(* CODESYS project Tc3_UnitTest.library
   Description: Twincat 3 unit test library
   Version: 1.0.0.4
   Title: Tc3_UnitTest
   Company: Zerlauth
   DocFormat: TcDocGen
   Placeholder: Tc3_UnitTest
   Author: www.peterzerlauth.com
   DefaultNamespace: Tc3_UnitTest

Project tree, tasks and I/O mapping:
  libraries: Tc2_Standard, * (Beckhoff Automation GmbH); Tc2_System, * (Beckhoff Automation GmbH); Tc2_Utilities, * (Beckhoff Automation GmbH); Tc3_JsonXml, * (Beckhoff Automation GmbH); Tc3_Module, * (Beckhoff Automation GmbH)
  Assert/
    data type E_AdsError
    data type E_Assert
    function block FB_Assert [ST]: M_Assert, M_Equals, M_Equals_Array_LREAL, M_Equals_Array_REAL, M_Equals_BOOL, M_Equals_BYTE, M_Equals_DINT, M_Equals_INT, M_Equals_LINT, M_Equals_LREAL, M_Equals_REAL, M_Equals_STRING, M_Equals_TIME, M_Equals_UDINT, M_Equals_UINT, M_Equals_ULINT, M_Equals_UXINT, M_Equals_WSTRING, M_Equals_XINT, M_Equals_XWORD, M_Error, M_Failure, M_IsTRUE, M_Passed, M_Reset, M_Skip
    interface I_Assert: M_Assert, M_Equals, M_Equals_Array_LREAL, M_Equals_Array_REAL, M_Equals_BOOL, M_Equals_BYTE, M_Equals_DINT, M_Equals_INT, M_Equals_LINT, M_Equals_LREAL, M_Equals_REAL, M_Equals_STRING, M_Equals_TIME, M_Equals_UDINT, M_Equals_UINT, M_Equals_ULINT, M_Equals_UXINT, M_Equals_WSTRING, M_Equals_XINT, M_Equals_XWORD, M_Error, M_Failure, M_IsTRUE, M_Passed, M_Reset, M_Skip
  Base/
    data type E_Base
    function F_GetCycleTime [ST]
    function F_GetName [ST]
    function block FB_Base [ST]: M_Aborted, M_Aborting, M_Execute, M_Init, M_Request, M_Starting, M_Stopped, M_Stopping, P_State
    interface I_Base: M_Request, P_State
  File/
    function block FB_File [ST]: M_Append, M_AppendLine, M_Close, M_Create, M_Delete, M_Load, M_Open, M_Read, M_Write, P_Error
    interface I_File: M_Append, M_AppendLine, M_Close, M_Create, M_Delete, M_Load, M_Open, M_Read, M_Write, P_Error
  List/
    Builder/
      function block FB_StringBuilder [ST]: FB_exit, M_Append, M_AppendBOOL, M_AppendINT, M_AppendREAL, M_Contains, M_Find, M_Insert, M_Reset, M_ToAny, M_ToString, P_Length
      interface I_StringBuilder: M_Append, M_AppendBOOL, M_AppendINT, M_AppendREAL, M_Contains, M_Find, M_Insert, M_Reset, M_ToAny, M_ToString, P_Length
    Object/
      function block FB_ListObject [ST]: FB_exit, M_Add, M_Clear, M_Find, M_Get, M_Index, M_Remove, P_Length
      interface I_ListObject: M_Add, M_Clear, M_Find, M_Get, M_Index, M_Remove, P_Length
      interface I_Object
    String/
      function block FB_ListSTRING [ST]: FB_exit, M_Add, M_Clear, M_Find, M_Index, M_Insert, M_Item, M_Remove, M_Set, P_Length
      interface I_ListSTRING: M_Add, M_Clear, M_Find, M_Index, M_Insert, M_Item, M_Remove, M_Set, P_Length
  Logger/
    data type E_LogLevel
    function block FB_Logger [ST]: M_Critical, M_Debug, M_Error, M_Info, M_Log, M_Warning, P_Settings
    function block FB_TcLogger [ST]: M_Critical, M_Debug, M_Error, M_Info, M_Log, M_Warning, P_Settings
    interface I_Logger: M_Critical, M_Debug, M_Error, M_Info, M_Log, M_Warning, P_Settings
    data type ST_LoggerSettings
  Property/
    function block FB_Property [ST]: M_Add, M_Reset, P_List
    interface I_Property: M_Add, M_Reset
  Testcase/
    data type E_Testcase
    data type ST_Testcase
  Testsuite/
    function block FB_Testsuite [ST]: M_Execute, M_Starting, M_Stopping, M_Testcase, P_Assert, P_File, P_List, P_Logger, P_Options, P_Parent, P_Property, P_Testcase
    interface I_Testsuite: P_File, P_List, P_Logger, P_Options, P_Parent, P_Testcase
    data type ST_Testsuite
    data type ST_TestsuiteOptions
  Testsuites/
    function block FB_Testsuites [ST]: M_Add, M_Execute, M_Starting, M_Stopping, P_Data, P_List, P_Options, P_Property
    interface I_Testsuites: P_Data, P_List, P_Options, P_Property
    data type ST_Testsuites
    data type ST_TestsuitesOptions
  Version/
    global variables Global_Version
*)

// Assert/E_AdsError
{attribute 'qualified_only'}
{attribute 'to_string'}
TYPE E_AdsError :
(
	NOERR:= 0,
	ROUTER_NOLOCKEDMEMORY:= 1280,
	ROUTER_RESIZEMEMORY:= 1281,
	ROUTER_MAILBOXFULL:= 1282,
	ROUTER_DEBUGBOXFULL:= 1283,
	ROUTER_UNKNOWNPORTTYPE:= 1284,
	ROUTER_NOTINITIALIZED:= 1285,
	ROUTER_PORTALREADYINUSE:= 1286,
	ROUTER_NOTREGISTERED:= 1287,
	ROUTER_NOMOREQUEUES:= 1288,
	ROUTER_INVALIDPORT:= 1289,
	ROUTER_NOTACTIVATED:= 1290,
	ROUTER_FRAGMENTBOXFULL:= 1291,
	ROUTER_FRAGMENTTIMEOUT:= 1292,
	ROUTER_TOBEREMOVED:= 1293,
	DEVICE_ERROR:= 1792,
	DEVICE_SRVNOTSUPP:= 1793,
	DEVICE_INVALIDGRP:= 1794,
	DEVICE_INVALIDOFFSET:= 1795,
	DEVICE_INVALIDACCESS:= 1796,
	DEVICE_INVALIDSIZE:= 1797,
	DEVICE_INVALIDDATA:= 1798,
	DEVICE_NOTREADY:= 1799,
	DEVICE_BUSY:= 1800,
	DEVICE_INVALIDCONTEXT:= 1801,
	DEVICE_NOMEMORY:= 1802,
	DEVICE_INVALIDPARM:= 1803,
	DEVICE_NOTFOUND:= 1804,
	DEVICE_SYNTAX:= 1805,
	DEVICE_INCOMPATIBLE:= 1806,
	DEVICE_EXISTS:= 1807,
	DEVICE_SYMBOLNOTFOUND:= 1808,
	DEVICE_SYMBOLVERSIONINVALID:= 1809,
	DEVICE_INVALIDSTATE:= 1810,
	DEVICE_TRANSMODENOTSUPP:= 1811,
	DEVICE_NOTIFYHNDINVALID:= 1812,
	DEVICE_CLIENTUNKNOWN:= 1813,
	DEVICE_NOMOREHDLS:= 1814,
	DEVICE_INVALIDWATCHSIZE:= 1815,
	DEVICE_NOTINIT:= 1816,
	DEVICE_TIMEOUT:= 1817,
	DEVICE_NOINTERFACE:= 1818,
	DEVICE_INVALIDINTERFACE:= 1819,
	DEVICE_INVALIDCLSID:= 1820,
	DEVICE_INVALIDOBJID:= 1821,
	DEVICE_PENDING:= 1822,
	DEVICE_ABORTED:= 1823,
	DEVICE_WARNING:= 1824,
	DEVICE_INVALIDARRAYIDX:= 1825,
	DEVICE_SYMBOLNOTACTIVE:= 1826,
	DEVICE_ACCESSDENIED:= 1827,
	DEVICE_LICENSENOTFOUND:= 1828,
	DEVICE_LICENSEEXPIRED:= 1829,
	DEVICE_LICENSEEXCEEDED:= 1830,
	DEVICE_LICENSEINVALID:= 1831,
	DEVICE_LICENSESYSTEMID:= 1832,
	DEVICE_LICENSENOTIMELIMIT:= 1833,
	DEVICE_LICENSEFUTUREISSUE:= 1834,
	DEVICE_LICENSETIMETOLONG:= 1835,
	DEVICE_EXCEPTION:= 1836,
	DEVICE_LICENSEDUPLICATED:= 1837,
	CLIENT_ERROR:= 1856,
	CLIENT_INVALIDPARM:= 1857,
	CLIENT_LISTEMPTY:= 1858,
	CLIENT_VARUSED:= 1859,
	CLIENT_DUPLINVOKEID:= 1860,
	CLIENT_SYNCTIMEOUT:= 1861,
	CLIENT_W32ERROR:= 1862,
	CLIENT_TIMEOUTINVALID:= 1863,
	CLIENT_PORTNOTOPEN:= 1864,
	CLIENT_NOAMSADDR:= 1865,
	CLIENT_SYNCINTERNAL:= 1872,
	CLIENT_ADDHASH:= 1873,
	CLIENT_REMOVEHASH:= 1874,
	CLIENT_NOMORESYM:= 1875,
	CLIENT_SYNCRESINVALID:= 1876,
	CLIENT_SYNCPORTLOCKED:= 1877
)UDINT;
END_TYPE

// Assert/E_Assert
{attribute 'qualified_only'}
{attribute 'strict'}
TYPE E_Assert :
(
	Passed	:= 0,
	Failure	:= 1,
	Error	:= 2,
	Skipped	:= 3
)USINT;
END_TYPE

// Base/E_Base
{attribute 'qualified_only'}
{attribute 'strict'}
TYPE E_Base :
(
	{attribute 'hide'} 
	Init 	:= 0,
	Starting:= 2,	
	Execute	:= 3,
	Stopping:= 4,
	Aborting:= 5,
	Aborted	:= 6,
	Reset	:= 7,
	Stopped	:= 1
)USINT;
END_TYPE

// Logger/E_LogLevel
{attribute 'qualified_only'}
{attribute 'strict'}
TYPE E_LogLevel :
(
	Debug:=		0, 
    Info:= 		1, 
    Warning:= 	2, 
    Error:= 	3, 
    Critical:= 	4
);
END_TYPE

// Logger/ST_LoggerSettings
TYPE ST_LoggerSettings :
STRUCT
	eLogLevelMinimum:		E_LogLevel:= E_LogLevel.Debug;
	eLogLevelMaximum:		E_LogLevel:= E_LogLevel.Critical;
END_STRUCT
END_TYPE

// Testcase/E_Testcase
{attribute 'qualified_only'}
{attribute 'strict'}
TYPE E_Testcase :
(
	Init    := -32768,
	Start 	:= 0,
	Done	:= 32767
)INT;
END_TYPE

// Testcase/ST_Testcase
TYPE ST_Testcase :
STRUCT
	sName:				STRING(255);	//	name        The name of this test case, often the method name  
	sClassname:			STRING(255);	//	classname   The name of the parent class/folder, often the same as the suite's name
	nAssertions:		DINT; 			//	assertions  Number of assertions checked during test case execution  
	fTime:				LREAL;			//	time        Execution time of the test in seconds            
	sFile:				STRING(255);	//	file        Source code file of this test case              
	sLine:				STRING(255);	//	line        Source code line number of the start of this test case  
END_STRUCT
END_TYPE

// Testsuite/ST_Testsuite
TYPE ST_Testsuite :
STRUCT
	sName:				STRING(255):= 'testsuite'; 	// Name OF the entire test run
	nTests:				DINT;						// tests       Total number of tests in this suite          
	nFailures:			DINT;						// failures    Total number of failed tests in this suite   
	nErrors:			DINT;						// errors      Total number of errored tests in this suite 
	nSkipped:			DINT;						// skipped     Total number of skipped tests in this suite            
	nAssertions:		DINT;						// assertions  Total number of assertions for all tests in this suite  
	fTime: 				LREAL;						// time        Aggregated time of all tests in this file in seconds  (100ns)   
	sTimestamp:			STRING(39);					// timestamp   Date and time of when the test suite was executed (in ISO 8601 format)  
	sFile:				STRING(255);				// file        Source code file of this test suite
END_STRUCT
END_TYPE

// Testsuite/ST_TestsuiteOptions
TYPE ST_TestsuiteOptions :
STRUCT
		bAbortOnError:			BOOL;
END_STRUCT
END_TYPE

// Testsuites/ST_Testsuites
TYPE ST_Testsuites :
STRUCT
	sName:				STRING(255); 				// Name OF the entire test run
	nTests:				DINT;						// Total number of tests in this file
	nFailures:			dINT;						// Total number of failed tests in this file
	nErrors:			dINT;						// Total number of errored tests in this file
	nSkipped:			dINT;						// Total number of skipped tests in this file
	nAssertions:		dINT;						// Total number of assertions for all tests in this file
	fTime:				LREAL;						// Aggregated time of all tests in this file in seconds
	sTimestamp:			STRING(39);					// timestamp   Date and time of when the test suite was executed (in ISO 8601 format)
END_STRUCT
END_TYPE

// Testsuites/ST_TestsuitesOptions
TYPE ST_TestsuitesOptions :
STRUCT
	sFilePathName:		STRING(255):= 'C:\report.xml';		// as Property
END_STRUCT
END_TYPE

// Version/Global_Version
{attribute 'TcGenerated'}
{attribute 'no-analysis'}
{attribute 'linkalways'}
// This function has been automatically generated from the project information.
VAR_GLOBAL CONSTANT
	{attribute 'const_non_replaced'}
	stLibVersion_Tc3_UnitTest : ST_LibVersion := (iMajor := 1, iMinor := 0, iBuild := 0, iRevision := 4, nFlags := 0, sVersion := '1.0.0.4');
END_VAR

// Assert/FB_Assert
FUNCTION_BLOCK FB_Assert IMPLEMENTS I_Assert
VAR_INPUT
END_VAR
VAR_OUTPUT
	fbList:					FB_ListSTRING;
	nAssert:				DINT;
	nPassed:				DINT;
	nSkipped:				DINT;
	nFailures:				DINT;
	nErrors:				DINT;
END_VAR
VAR
	fbJson:					FB_JsonSaxWriter;
  	fbJsonDataType:			FB_JsonReadWriteDataType;
	fbBuilder:				FB_StringBuilder;
END_VAR

METHOD PUBLIC M_Assert
VAR_INPUT
END_VAR
IF nSkipped = 0 THEN
	nAssert:= nAssert + 1;
END_IF
END_METHOD

METHOD PUBLIC M_Equals : I_Assert
VAR_INPUT
	Expected:			ANY;			// Expected as udint
    Actual:				ANY;          	// Actual as udint
	Message:			STRING(255);   	// Message as string
END_VAR
VAR
	sJsonExpected:			STRING(2000);
	sJsonActual:			STRING(2000); 
	sDatatypeExpected:		STRING(255); 
	sDatatypeActual:		STRING(255);
END_VAR
M_Assert();

fbJson.ResetDocument();
sDatatypeExpected:= fbJsonDataType.GetDatatypeNameByAddress(nData:= DINT_TO_UDINT(Expected.diSize), pData:= Expected.pValue);
fbJsonDataType.AddJsonValueFromSymbol(fbJson, sDatatypeExpected, DINT_TO_UDINT(Expected.diSize), Expected.pValue);
fbJson.CopyDocument(sJsonExpected, SIZEOF(sJsonExpected));

fbJson.ResetDocument();
sDatatypeActual:= fbJsonDataType.GetDatatypeNameByAddress(nData:= DINT_TO_UDINT(Actual.diSize), pData:= Actual.pValue);
fbJsonDataType.AddJsonValueFromSymbol(fbJson, sDatatypeActual, DINT_TO_UDINT(Actual.diSize), Actual.pValue);
fbJson.CopyDocument(sJsonActual, SIZEOF(sJsonActual));

IF sDatatypeExpected <> sDatatypeActual THEN
	fbBuilder.M_Reset();
	fbBuilder.M_Append('Expected = ');
	fbBuilder.M_Append(sDatatypeExpected);
	fbBuilder.M_Append(' Actual = ');
	fbBuilder.M_Append(sDatatypeActual);
	M_Failure(fbBuilder.M_ToString(), Message);
ELSIF sJsonExpected <> sJsonActual THEN
	fbBuilder.M_Reset();
	fbBuilder.M_Append('Expected = ');
	fbBuilder.M_Append(sJsonExpected);
	fbBuilder.M_Append(' Actual = ');
	fbBuilder.M_Append(sJsonActual);
	M_Failure(fbBuilder.M_ToString(), Message);
END_IF
M_Equals:= THIS^;
END_METHOD

METHOD PUBLIC M_Equals_Array_LREAL : I_Assert
VAR_IN_OUT
	Expected:			ARRAY [*] OF LREAL;	// Expected as array of lreal
	Actual:				ARRAY [*] OF LREAL;	// Actual as array of lreal
END_VAR                                    
VAR_INPUT                                  
	Tolerance:			LREAL;              // Tolerance as lreal
	Message:			STRING(255);		// Message as string
END_VAR

VAR
	nIndex:				DINT;
END_VAR
M_Equals_Array_LREAL:= THIS^;
M_Assert();
IF LOWER_BOUND(Expected, 1) <> LOWER_BOUND(Actual, 1) THEN
	M_Failure('', Message);
ELSIF UPPER_BOUND(Expected, 1) <> UPPER_BOUND(Actual, 1) THEN
	M_Failure('', Message);
ELSE
	FOR nIndex:= LOWER_BOUND(Expected, 1) TO UPPER_BOUND(Expected, 1) DO
		IF ABS(Expected[nIndex] - Actual[nIndex]) > ABS(Tolerance) THEN	
			fbBuilder.M_Reset();
			fbBuilder.M_Append('Index = [');
			fbBuilder.M_Append(DINT_TO_STRING(nIndex));
			fbBuilder.M_Append('] Expected = ]');
			fbBuilder.M_Append(LREAL_TO_STRING(Expected[nIndex]));
			fbBuilder.M_Append('] Actual = [');
			fbBuilder.M_Append(LREAL_TO_STRING(Actual[nIndex]));
			fbBuilder.M_Append('] Tolerance = ]');
			fbBuilder.M_Append(LREAL_TO_STRING(Tolerance));
			fbBuilder.M_Append(']');
			M_Failure(fbBuilder.M_ToString(), Message);
			RETURN;
		END_IF
	END_FOR
	M_Passed();
END_IF
END_METHOD

METHOD PUBLIC M_Equals_Array_REAL : I_Assert
VAR_IN_OUT
	Expected:			ARRAY [*] OF REAL;	// Expected as array of real
	Actual:				ARRAY [*] OF REAL;	// Actual as array of real
END_VAR                                   
VAR_INPUT                                 
	Tolerance:			REAL;             	// Tolerance as real
	Message:			STRING(255);      	// Message as string
END_VAR

VAR
	nIndex:				DINT;
END_VAR
M_Equals_Array_REAL:= THIS^;
M_Assert();
IF LOWER_BOUND(Expected, 1) <> LOWER_BOUND(Actual, 1) THEN
	M_Failure('', Message);
ELSIF UPPER_BOUND(Expected, 1) <> UPPER_BOUND(Actual, 1) THEN
	M_Failure('', Message);
ELSE
	FOR nIndex:= LOWER_BOUND(Expected, 1) TO UPPER_BOUND(Expected, 1) DO
		IF ABS(Expected[nIndex] - Actual[nIndex]) > ABS(Tolerance) THEN	
			fbBuilder.M_Reset();
			fbBuilder.M_Append('Index = [');
			fbBuilder.M_Append(DINT_TO_STRING(nIndex));
			fbBuilder.M_Append('] Expected = ]');
			fbBuilder.M_Append(REAL_TO_STRING(Expected[nIndex]));
			fbBuilder.M_Append('] Actual = "');
			fbBuilder.M_Append(REAL_TO_STRING(Actual[nIndex]));
			fbBuilder.M_Append('] Tolerance = [');
			fbBuilder.M_Append(REAL_TO_STRING(Tolerance));
			fbBuilder.M_Append(']');
			M_Failure(fbBuilder.M_ToString(), Message);
			RETURN;
		END_IF
	END_FOR
	M_Passed();
END_IF
END_METHOD

METHOD PUBLIC M_Equals_BOOL : I_Assert
VAR_INPUT
	Expected:			BOOL;				// Expected as bool
    Actual:				BOOL;           	// Actual as bool
	Message:			STRING(255);    	// Message as string
END_VAR
M_Assert();
IF Expected = Actual THEN
	M_Passed();
ELSE
	fbBuilder.M_Reset();
	fbBuilder.M_Append('Expected = [');
	fbBuilder.M_Append(BOOL_TO_STRING(Expected));
	fbBuilder.M_Append('] Actual = [');
	fbBuilder.M_Append(BOOL_TO_STRING(Actual));
	fbBuilder.M_Append(']');
	M_Failure(fbBuilder.M_ToString(), Message);
END_IF
M_Equals_BOOL:= THIS^;
END_METHOD

METHOD PUBLIC M_Equals_BYTE : I_Assert
VAR_INPUT
	Expected:			BYTE;			// Expected as byte
    Actual:				BYTE;           // Actual as byte
	Message:			STRING(255);    // Message as string
END_VAR
M_Assert();
IF Expected = Actual THEN
	M_Passed();
ELSE
	fbBuilder.M_Reset();
	fbBuilder.M_Append('Expected = [');
	fbBuilder.M_Append(BYTE_TO_STRING(Expected));
	fbBuilder.M_Append('] Actual = [');
	fbBuilder.M_Append(BYTE_TO_STRING(Actual));
	fbBuilder.M_Append(']');
	M_Failure(fbBuilder.M_ToString(), Message);
END_IF
M_Equals_BYTE:= THIS^;
END_METHOD

METHOD PUBLIC M_Equals_DINT : I_Assert
VAR_INPUT
	Expected:			DINT;			// Expected as dint
    Actual:				DINT;           // Actual as dint
	Message:			STRING(255);    // Message as string
END_VAR
M_Assert();
IF Expected = Actual THEN
	M_Passed();
ELSE
	fbBuilder.M_Reset();
	fbBuilder.M_Append('Expected = [');
	fbBuilder.M_Append(DINT_TO_STRING(Expected));
	fbBuilder.M_Append('] Actual = [');
	fbBuilder.M_Append(DINT_TO_STRING(Actual));
	fbBuilder.M_Append(']');
	M_Failure(fbBuilder.M_ToString(), Message);
END_IF
M_Equals_DINT:= THIS^;
END_METHOD

METHOD PUBLIC M_Equals_INT : I_Assert
VAR_INPUT
	Expected:			INT;			// Expected as int
    Actual:				INT;            // Actual as int
	Message:			STRING(255);    // Message as string
END_VAR
M_Assert();
IF Expected = Actual THEN
	M_Passed();
ELSE
	fbBuilder.M_Reset();
	fbBuilder.M_Append('Expected = [');
	fbBuilder.M_Append(INT_TO_STRING(Expected));
	fbBuilder.M_Append('] Actual = [');
	fbBuilder.M_Append(INT_TO_STRING(Actual));
	fbBuilder.M_Append(']');
	M_Failure(fbBuilder.M_ToString(), Message);
END_IF
M_Equals_INT:= THIS^;
END_METHOD

METHOD PUBLIC M_Equals_LINT : I_Assert
VAR_INPUT
	Expected:			LINT;			// Expected as lint
    Actual:				LINT;           // Actual as lint
	Message:			STRING(255);    // Message as string
END_VAR
M_Assert();
IF Expected = Actual THEN
	M_Passed();
ELSE
	fbBuilder.M_Reset();
	fbBuilder.M_Append('Expected = [');
	fbBuilder.M_Append(LINT_TO_STRING(Expected));
	fbBuilder.M_Append('] Actual = [');
	fbBuilder.M_Append(LINT_TO_STRING(Actual));
	fbBuilder.M_Append(']');
	M_Failure(fbBuilder.M_ToString(), Message);
END_IF
M_Equals_LINT:= THIS^;
END_METHOD

METHOD PUBLIC M_Equals_LREAL : I_Assert
VAR_INPUT
	Expected:			LREAL;				// Expected as lreal
    Actual:				LREAL;              // Actual as lreal
	Tolerance:			LREAL;             	// Tolerance as lreal         
	Message:			STRING(255);		// Message as string
END_VAR
M_Assert();
IF LrealIsNaN(Expected) THEN
	M_Failure('', Concat('Expected is NaN', Message));
ELSIF LrealIsNaN(Actual) THEN
	M_Failure('', Concat('Actual is NaN', Message));	
ELSIF LrealIsNaN(Tolerance) THEN
	M_Failure('', Concat('Tolerance is NaN', Message));	
ELSIF ABS(Expected - Actual) <= ABS(Tolerance) THEN
	M_Passed();
ELSE
	fbBuilder.M_Reset();
	fbBuilder.M_Append('Expected = [');
	fbBuilder.M_Append(LREAL_TO_STRING(Expected));
	fbBuilder.M_Append('] Actual = [');
	fbBuilder.M_Append(LREAL_TO_STRING(Actual));
	fbBuilder.M_Append('] Tolerance = [');
	fbBuilder.M_Append(LREAL_TO_STRING(Tolerance));
	fbBuilder.M_Append(']');
	M_Failure(fbBuilder.M_ToString(), Message);
END_IF
M_Equals_LREAL:= THIS^;
END_METHOD

METHOD PUBLIC M_Equals_REAL : I_Assert
VAR_INPUT
	Expected:			REAL;			// Expected as real
    Actual:				REAL;           // Actual as real
	Tolerance:			REAL;           // Tolerance as real    
	Message:			STRING(255);    // Message as string
END_VAR
M_Assert();
IF RealIsNaN(Expected) THEN
	M_Failure('', Concat('Expected is NaN', Message));
ELSIF RealIsNaN(Actual) THEN
	M_Failure('', Concat('Actual is NaN', Message));	
ELSIF RealIsNaN(Tolerance) THEN
	M_Failure('', Concat('Tolerance is NaN', Message));	
ELSIF ABS(Expected - Actual) <= ABS(Tolerance) THEN
	M_Passed();
ELSE
	fbBuilder.M_Reset();
	fbBuilder.M_Append('Expected = [');
	fbBuilder.M_Append(LREAL_TO_STRING(Expected));
	fbBuilder.M_Append('] Actual = [');
	fbBuilder.M_Append(LREAL_TO_STRING(Actual));
	fbBuilder.M_Append('] Tolerance = [');
	fbBuilder.M_Append(LREAL_TO_STRING(Tolerance));
	fbBuilder.M_Append(']');
	M_Failure(fbBuilder.M_ToString(), Message);
END_IF
M_Equals_REAL:= THIS^;
END_METHOD

METHOD PUBLIC M_Equals_STRING : I_Assert
VAR_INPUT
	Expected:			STRING(255);		// Expected as string
    Actual:				STRING(255);        // Actual as string
	Message:			STRING(255);      	// Message as string  
END_VAR
M_Assert();
IF Expected = Actual THEN
	M_Passed();
ELSE
	fbBuilder.M_Reset();
	fbBuilder.M_Append('Expected = [');
	fbBuilder.M_Append(Expected);
	fbBuilder.M_Append('] Actual = [');
	fbBuilder.M_Append(Actual);
	fbBuilder.M_Append(']');
	M_Failure(fbBuilder.M_ToString(), Message);
END_IF
M_Equals_STRING:= THIS^;
END_METHOD

METHOD PUBLIC M_Equals_TIME : I_Assert
VAR_INPUT
	Expected:			TIME;				// Expected as time
    Actual:				TIME;               // Actual as time
	Tolerance:			TIME;               // Tolerance as time    
	Message:			STRING(255);        // Message as string
END_VAR
M_Assert();
IF ABS(Expected - Actual) <= ABS(Tolerance) THEN
	M_Passed();
ELSE
	fbBuilder.M_Reset();
	fbBuilder.M_Append('Expected = [');
	fbBuilder.M_Append(TIME_TO_STRING(Expected));
	fbBuilder.M_Append('] Actual = [');
	fbBuilder.M_Append(TIME_TO_STRING(Actual));
	fbBuilder.M_Append('] Tolerance = [');
	fbBuilder.M_Append(TIME_TO_STRING(Tolerance));
	fbBuilder.M_Append(']');
	M_Failure(fbBuilder.M_ToString(), Message);
END_IF
M_Equals_TIME:= THIS^;
END_METHOD

METHOD PUBLIC M_Equals_UDINT : I_Assert
VAR_INPUT
	Expected:			UDINT;			// Expected as udint
    Actual:				UDINT;          // Actual as udint
	Message:			STRING(255);   	// Message as string
END_VAR
M_Assert();
IF Expected = Actual THEN
	M_Passed();
ELSE
	fbBuilder.M_Reset();
	fbBuilder.M_Append('Expected = [');
	fbBuilder.M_Append(UDINT_TO_STRING(Expected));
	fbBuilder.M_Append('] Actual = [');
	fbBuilder.M_Append(UDINT_TO_STRING(Actual));
	fbBuilder.M_Append(']');
	M_Failure(fbBuilder.M_ToString(), Message);
END_IF
M_Equals_UDINT:= THIS^;
END_METHOD

METHOD PUBLIC M_Equals_UINT : I_Assert
VAR_INPUT
	Expected:			UINT;			// Expected as uint
    Actual:				UINT;           // Actual as uint
	Message:			STRING(255);    // Message as string
END_VAR
M_Assert();
IF Expected = Actual THEN
	M_Passed();
ELSE
	fbBuilder.M_Reset();
	fbBuilder.M_Append('Expected = [');
	fbBuilder.M_Append(UINT_TO_STRING(Expected));
	fbBuilder.M_Append('] Actual = [');
	fbBuilder.M_Append(UINT_TO_STRING(Actual));
	fbBuilder.M_Append(']');
	M_Failure(fbBuilder.M_ToString(), Message);
END_IF
M_Equals_UINT:= THIS^;
END_METHOD

METHOD PUBLIC M_Equals_ULINT : I_Assert
VAR_INPUT
	Expected:			ULINT;			// Expected as ulint
    Actual:				ULINT;          // Actual as ulint
	Message:			STRING(255);    // Message as string
END_VAR
M_Assert();
IF Expected = Actual THEN
	M_Passed();
ELSE
	fbBuilder.M_Reset();
	fbBuilder.M_Append('Expected = [');
	fbBuilder.M_Append(ULINT_TO_STRING(Expected));
	fbBuilder.M_Append('] Actual = [');
	fbBuilder.M_Append(ULINT_TO_STRING(Actual));
	fbBuilder.M_Append(']');
	M_Failure(fbBuilder.M_ToString(), Message);
END_IF
M_Equals_ULINT:= THIS^;
END_METHOD

METHOD PUBLIC M_Equals_UXINT : I_Assert
VAR_INPUT
	Expected:			UXINT;			// Expected as udint
    Actual:				UXINT;          // Actual as udint
	Message:			STRING(255);   	// Message as string
END_VAR
M_Assert();
IF Expected = Actual THEN
	M_Passed();
ELSE
	fbBuilder.M_Reset();
	fbBuilder.M_Append('Expected = [');
	fbBuilder.M_Append(TO_STRING(Expected));
	fbBuilder.M_Append('] Actual = [');
	fbBuilder.M_Append(TO_STRING(Actual));
	fbBuilder.M_Append(']');
	M_Failure(fbBuilder.M_ToString(), Message);
END_IF
M_Equals_UXINT:= THIS^;
END_METHOD

METHOD PUBLIC M_Equals_WSTRING : I_Assert
VAR_INPUT
	Expected:			WSTRING(255);		// Expected as wstring
    Actual:				WSTRING(255);       // Actual as wstring
	Message:			STRING(255);        // Message as string
END_VAR
M_Assert();
IF Expected = Actual THEN
	M_Passed();
ELSE
	fbBuilder.M_Reset();
	fbBuilder.M_Append('Expected = [');
	fbBuilder.M_Append(WSTRING_TO_STRING(Expected));
	fbBuilder.M_Append('] Actual = [');
	fbBuilder.M_Append(WSTRING_TO_STRING(Actual));
	fbBuilder.M_Append(']');
	M_Failure(fbBuilder.M_ToString(), Message);
END_IF
M_Equals_WSTRING:= THIS^;
END_METHOD

METHOD PUBLIC M_Equals_XINT : I_Assert
VAR_INPUT
	Expected:			XINT;			// Expected as udint
    Actual:				XINT;          // Actual as udint
	Message:			STRING(255);   	// Message as string
END_VAR
M_Assert();
IF Expected = Actual THEN
	M_Passed();
ELSE
	fbBuilder.M_Reset();
	fbBuilder.M_Append('Expected = [');
	fbBuilder.M_Append(TO_STRING(Expected));
	fbBuilder.M_Append('] Actual = [');
	fbBuilder.M_Append(TO_STRING(Actual));
	fbBuilder.M_Append(']');
	M_Failure(fbBuilder.M_ToString(), Message);
END_IF
M_Equals_XINT:= THIS^;
END_METHOD

METHOD PUBLIC M_Equals_XWORD : I_Assert
VAR_INPUT
	Expected:			XWORD;			// Expected as udint
    Actual:				XWORD;          // Actual as udint
	Message:			STRING(255);   	// Message as string
END_VAR
M_Assert();
IF Expected = Actual THEN
	M_Passed();
ELSE
	fbBuilder.M_Reset();
	fbBuilder.M_Append('Expected = [');
	fbBuilder.M_Append(TO_STRING(Expected));
	fbBuilder.M_Append('] Actual = [');
	fbBuilder.M_Append(TO_STRING(Actual));
	fbBuilder.M_Append(']');
	M_Failure(fbBuilder.M_ToString(), Message);
END_IF
M_Equals_XWORD:= THIS^;
END_METHOD

METHOD PUBLIC M_Error
VAR_INPUT
	Data:				STRING(255);
	Message:			STRING(255);
END_VAR
IF nSkipped = 0 THEN
	fbBuilder.M_Reset();
	fbBuilder.M_Append('$T$T$T<error message="');
	fbBuilder.M_Append(Message);
	fbBuilder.M_Append('" type="ArithmeticError">');
	fbBuilder.M_Append(Data);	
	fbBuilder.M_Append('</error>');
	fbList.M_Add(fbBuilder.M_ToString());
	nErrors:= nErrors + 1;
END_IF
END_METHOD

METHOD PUBLIC M_Failure
VAR_INPUT
	Data:				STRING(255);
	Message:			STRING(255);
END_VAR
IF nSkipped = 0 THEN
	fbBuilder.M_Reset();
	fbBuilder.M_Append('$T$T$T<failure message="');
	fbBuilder.M_Append(Message);
	fbBuilder.M_Append('" type="AssertionError">');
	fbBuilder.M_Append(Data);
	fbBuilder.M_Append('</failure>');
	fbList.M_Add(fbBuilder.M_ToString());
	nFailures:= nFailures + 1;
END_IF
END_METHOD

METHOD PUBLIC M_IsTRUE : I_Assert
VAR_INPUT
    Actual:				BOOL;				// Actual as bool
	Message:			STRING(255);        // Message as string
END_VAR
M_Assert();
IF Actual THEN
	M_Passed();
ELSE
	M_Failure('Actual = "FALSE"', Message);
END_IF
M_IsTRUE:= THIS^;
END_METHOD

METHOD PUBLIC M_Passed
VAR_INPUT
END_VAR
IF nSkipped = 0 THEN
	nPassed:= nPassed + 1;
END_IF
END_METHOD

METHOD PUBLIC M_Reset : I_Assert
VAR_INPUT
END_VAR
fbList.M_Clear();
nAssert:= 0;
nPassed:= 0;
nSkipped:= 0;
nFailures:= 0;
nErrors:= 0;
M_Reset:= THIS^;
END_METHOD

METHOD PUBLIC M_Skip
VAR_INPUT
	Message:			STRING(255);	// Message as string
END_VAR
fbList.M_Clear();
nAssert:= 0;
nPassed:= 0;
nFailures:= 0;
nErrors:= 0;
fbBuilder.M_Reset();
fbBuilder.M_Append('$T$T$T<skipped message="');
fbBuilder.M_Append(Message);
fbBuilder.M_Append('" />');
fbList.M_Add(fbBuilder.M_ToString());
nSkipped:= nSkipped + 1;
END_METHOD

END_FUNCTION_BLOCK

// Assert/I_Assert
INTERFACE I_Assert

METHOD PUBLIC M_Assert
VAR_INPUT
END_VAR
END_METHOD

METHOD PUBLIC M_Equals : I_Assert
VAR_INPUT
	Expected:			ANY;			// Expected as udint
    Actual:				ANY;          // Actual as udint
	Message:			STRING(255);   	// Message as string
END_VAR
END_METHOD

METHOD PUBLIC M_Equals_Array_LREAL : I_Assert
VAR_IN_OUT
	Expected:			ARRAY [*] OF LREAL;	// Expected as array of lreal
	Actual:				ARRAY [*] OF LREAL;	// Actual as array of lreal
END_VAR                                    
VAR_INPUT                                  
	Tolerance:			LREAL;              // Tolerance as lreal
	Message:			STRING(255);		// Message as string
END_VAR
END_METHOD

METHOD PUBLIC M_Equals_Array_REAL : I_Assert
VAR_IN_OUT
	Expected:			ARRAY [*] OF REAL;	// Expected as array of real
	Actual:				ARRAY [*] OF REAL;	// Actual as array of real
END_VAR                                   
VAR_INPUT                                 
	Tolerance:			REAL;             	// Tolerance as real
	Message:			STRING(255);      	// Message as string
END_VAR
END_METHOD

METHOD PUBLIC M_Equals_BOOL : I_Assert
VAR_INPUT
	Expected:			BOOL;				// Expected as bool
    Actual:				BOOL;           	// Actual as bool
	Message:			STRING(255);    	// Message as string
END_VAR
END_METHOD

METHOD PUBLIC M_Equals_BYTE : I_Assert
VAR_INPUT
	Expected:			BYTE;			// Expected as byte
    Actual:				BYTE;           // Actual as byte
	Message:			STRING(255);    // Message as string
END_VAR
END_METHOD

METHOD PUBLIC M_Equals_DINT : I_Assert
VAR_INPUT
	Expected:			DINT;			// Expected as dint
    Actual:				DINT;           // Actual as dint
	Message:			STRING(255);    // Message as string
END_VAR
END_METHOD

METHOD PUBLIC M_Equals_INT : I_Assert
VAR_INPUT
	Expected:			INT;			// Expected as int
    Actual:				INT;            // Actual as int
	Message:			STRING(255);    // Message as string
END_VAR
END_METHOD

METHOD PUBLIC M_Equals_LINT : I_Assert
VAR_INPUT
	Expected:			LINT;			// Expected as lint
    Actual:				LINT;           // Actual as lint
	Message:			STRING(255);    // Message as string
END_VAR
END_METHOD

METHOD PUBLIC M_Equals_LREAL : I_Assert
VAR_INPUT
	Expected:			LREAL;				// Expected as lreal
    Actual:				LREAL;              // Actual as lreal
	Tolerance:			LREAL;             	// Tolerance as lreal         
	Message:			STRING(255);		// Message as string
END_VAR
END_METHOD

METHOD PUBLIC M_Equals_REAL : I_Assert
VAR_INPUT
	Expected:			REAL;			// Expected as real
    Actual:				REAL;           // Actual as real
	Tolerance:			REAL;           // Tolerance as real    
	Message:			STRING(255);    // Message as string
END_VAR
END_METHOD

METHOD PUBLIC M_Equals_STRING : I_Assert
VAR_INPUT
	Expected:			STRING(255);		// Expected as string
    Actual:				STRING(255);        // Actual as string
	Message:			STRING(255);      	// Message as string  
END_VAR
END_METHOD

METHOD PUBLIC M_Equals_TIME : I_Assert
VAR_INPUT
	Expected:			TIME;				// Expected as time
    Actual:				TIME;               // Actual as time
	Tolerance:			TIME;               // Tolerance as time    
	Message:			STRING(255);        // Message as string
END_VAR
END_METHOD

METHOD PUBLIC M_Equals_UDINT : I_Assert
VAR_INPUT
	Expected:			UDINT;			// Expected as udint
    Actual:				UDINT;          // Actual as udint
	Message:			STRING(255);   	// Message as string
END_VAR
END_METHOD

METHOD PUBLIC M_Equals_UINT : I_Assert
VAR_INPUT
	Expected:			UINT;			// Expected as uint
    Actual:				UINT;           // Actual as uint
	Message:			STRING(255);    // Message as string
END_VAR
END_METHOD

METHOD PUBLIC M_Equals_ULINT : I_Assert
VAR_INPUT
	Expected:			ULINT;			// Expected as ulint
    Actual:				ULINT;          // Actual as ulint
	Message:			STRING(255);    // Message as string
END_VAR
END_METHOD

METHOD PUBLIC M_Equals_UXINT : I_Assert
VAR_INPUT
	Expected:			UXINT;			// Expected as udint
    Actual:				UXINT;          // Actual as udint
	Message:			STRING(255);   	// Message as string
END_VAR
END_METHOD

METHOD PUBLIC M_Equals_WSTRING : I_Assert
VAR_INPUT
	Expected:			WSTRING(255);		// Expected as wstring
    Actual:				WSTRING(255);       // Actual as wstring
	Message:			STRING(255);        // Message as string
END_VAR
END_METHOD

METHOD PUBLIC M_Equals_XINT : I_Assert
VAR_INPUT
	Expected:			XINT;			// Expected as udint
    Actual:				XINT;          // Actual as udint
	Message:			STRING(255);   	// Message as string
END_VAR
END_METHOD

METHOD PUBLIC M_Equals_XWORD : I_Assert
VAR_INPUT
	Expected:			XWORD;			// Expected as udint
    Actual:				XWORD;          // Actual as udint
	Message:			STRING(255);   	// Message as string
END_VAR
END_METHOD

METHOD PUBLIC M_Error
VAR_INPUT
	Data:				STRING(255);
	Message:			STRING(255);
END_VAR
END_METHOD

METHOD PUBLIC M_Failure
VAR_INPUT
	Data:				STRING(255);
	Message:			STRING(255);
END_VAR
END_METHOD

METHOD PUBLIC M_IsTRUE : I_Assert
VAR_INPUT
    Actual:				BOOL;				// Actual as bool
	Message:			STRING(255);        // Message as string
END_VAR
END_METHOD

METHOD PUBLIC M_Passed
VAR_INPUT
END_VAR
END_METHOD

METHOD PUBLIC M_Reset : I_Assert
VAR_INPUT
END_VAR
END_METHOD

METHOD PUBLIC M_Skip
VAR_INPUT
	Message:			STRING(255);	// Message as string
END_VAR
END_METHOD

END_INTERFACE

// List/String/FB_ListSTRING
{attribute 'no_explicit_call'} 
FUNCTION_BLOCK PUBLIC FB_ListSTRING IMPLEMENTS I_ListSTRING
VAR
	pList: 			POINTER TO STRING(255);
	nLength:		DINT;
	aList:			POINTER TO POINTER TO ARRAY [0..100] OF STRING(255):=ADR(pList);
END_VAR

METHOD FB_exit : BOOL
VAR_INPUT
	bInCopyCode : BOOL; // if TRUE, the exit method is called for exiting an instance that is copied afterwards (online change).
END_VAR
M_Clear();
END_METHOD

METHOD M_Add : BOOL
VAR_INPUT
	Value:		STRING(255);
END_VAR
VAR
	pOldList: 	POINTER TO STRING(255);
END_VAR
// First Item
IF pList = 0 THEN
	nLength:= nLength + 1;
	pList:= __NEW(POINTER TO STRING(255), SIZEOF(STRING(255)));
ELSE
	// backup 
	pOldList:= pList;
	// new Length
	nLength:= nLength + 1;
	// new pointer
	pList:= __NEW(POINTER TO STRING(255),DINT_TO_UDINT(SIZEOF(STRING(255)) * nLength));
	// restore
	Memcpy(pList,pOldList, DINT_TO_UDINT(SIZEOF(STRING(255)) *(nLength -1)));
	// delete old
	__DELETE(pOldList);
END_IF

// add new Object
IF pList = 0 THEN
	RETURN;
END_IF
pList[nLength-1]:= Value;
M_Add:= TRUE;
END_METHOD

METHOD M_Clear : BOOL
IF pList <> 0 THEN
	nLength:= 0;
	__DELETE(pList);
	M_Clear:= TRUE;
END_IF
END_METHOD

METHOD M_Find : DINT
VAR_INPUT
	Value:		STRING(255);
END_VAR
VAR
	nIndex: 	UINT;
END_VAR
// Object already in List
M_Find := -1;
WHILE nIndex < nLength DO
    IF pList[nIndex] = Value THEN
        M_Find := nIndex;
        RETURN;
    END_IF
	nIndex := nIndex + 1;
END_WHILE
END_METHOD

METHOD M_Index : DINT
VAR_INPUT
	Value:	STRING(255);
END_VAR
VAR
	nIndex: 	DINT;
END_VAR
// Object already in List
M_Index := -1;
WHILE nIndex < nLength DO
  IF pList[nIndex] = Value THEN
        M_Index := nIndex;
        RETURN;
    END_IF
	nIndex := nIndex + 1;
END_WHILE
END_METHOD

METHOD PUBLIC M_Insert : BOOL
VAR_INPUT
	Position:		DINT;
	Value:			STRING(255);
END_VAR
VAR
	pOldList: 		POINTER TO STRING(255);
END_VAR
IF nLength > Position THEN
	// backup 
	pOldList:= pList;
	// new Length
	nLength:= nLength + 1;
	// new pointer
	pList:= __NEW(POINTER TO STRING(255),DINT_TO_UDINT(SIZEOF(STRING(255)) * nLength));
	// restore
	Memcpy(pList, pOldList, DINT_TO_UDINT(SIZEOF(STRING(255)) *(nLength -1)));
	MemMove(pList + DINT_TO_UDINT(SIZEOF(STRING(255)) * (Position + 1)), pList + DINT_TO_UDINT(SIZEOF(STRING(255)) * Position), DINT_TO_UDINT(SIZEOF(STRING(255)) * (nLength - Position + 1)));
	// delete old
	__DELETE(pOldList);
ELSE
	M_Insert:= FALSE;	
	RETURN;
END_IF
// add new Object
pList[Position]:= Value;
M_Insert:= TRUE;
END_METHOD

METHOD M_Item : STRING(255)
VAR_INPUT
	Index: 	DINT;
END_VAR
IF Index < (nLength) THEN
	M_Item:= pList[Index];
END_IF
END_METHOD

METHOD M_Remove : BOOL
VAR_INPUT
	Position:			DINT;
END_VAR
VAR
	pOldList:			POINTER TO STRING(255);
END_VAR
// First Item
IF nLength >= Position THEN
	// backup 
	pOldList:= pList;
	// new Length
	nLength:= nLength -1;
	// new pointer
	pList:= __NEW(POINTER TO STRING(255),DINT_TO_UDINT(SIZEOF(STRING(255)) * nLength));
	// restore lower part
	Memcpy(pList,pOldList, SIZEOF(POINTER TO STRING(255)) * DINT_TO_UDINT(Position));
	//pList[nPosition]:= iObject;
	Memcpy(pList + (SIZEOF(STRING(255))*Position),pOldList + (SIZEOF(STRING(255))*(Position + 1)), SIZEOF(STRING(255)) * DINT_TO_UDINT(nLength - Position));
	// delete old
	__DELETE(pOldList);
ELSE
	M_Remove:= FALSE;	
	RETURN;
END_IF
M_Remove:= TRUE;
END_METHOD

METHOD PUBLIC M_Set : BOOL
VAR_INPUT
	Index:			DINT;
	Value:			STRING(255);
END_VAR
IF Index < (nLength) THEN
	pList[Index]:= Value;
END_IF
END_METHOD

PROPERTY P_Length : DINT
GET
P_Length:= nLength;
END_GET
END_PROPERTY

END_FUNCTION_BLOCK

// List/String/I_ListSTRING
INTERFACE I_ListSTRING

METHOD M_Add : BOOL
VAR_INPUT
	Value:		STRING(255);
END_VAR
END_METHOD

METHOD M_Clear : BOOL
END_METHOD

METHOD M_Find : DINT
VAR_INPUT
	Value:		STRING(255);
END_VAR
END_METHOD

METHOD M_Index : DINT
VAR_INPUT
	Value:	STRING(255);
END_VAR
END_METHOD

METHOD PUBLIC M_Insert : BOOL
VAR_INPUT
	Position:		DINT;
	Value:			STRING(255);
END_VAR
END_METHOD

METHOD M_Item : STRING(255)
VAR_INPUT
	Index: 	DINT;
END_VAR
END_METHOD

METHOD M_Remove : BOOL
VAR_INPUT
	Position:			DINT;
END_VAR
END_METHOD

METHOD PUBLIC M_Set : BOOL
VAR_INPUT
	Index:			DINT;
	Value:			STRING(255);
END_VAR
END_METHOD

PROPERTY P_Length : DINT
GET
END_GET
END_PROPERTY

END_INTERFACE

// List/Builder/FB_StringBuilder
{attribute 'no_explicit_call'}
FUNCTION_BLOCK FB_StringBuilder IMPLEMENTS I_StringBuilder
VAR_INPUT
END_VAR
VAR_OUTPUT
END_VAR
VAR
	pString:		POINTER TO STRING(1);
	aList:			POINTER TO POINTER TO STRING(1000):= ADR(pString);
	nLength:		UDINT;
END_VAR

METHOD FB_exit : BOOL
VAR_INPUT
	bInCopyCode : BOOL; // if TRUE, the exit method is called for exiting an instance that is copied afterwards (online change).
END_VAR
M_Reset();
END_METHOD

METHOD M_Append : I_StringBuilder
VAR_INPUT
	Value	: STRING(255);
END_VAR
VAR
	pValue: 	POINTER TO STRING(1):=ADR(Value);
	nValue:		UDINT:= LEN2(pValue);
	pOldList:	POINTER TO STRING(1):= pString;
END_VAR
// First Item
IF pString = 0 THEN
	nLength:= nValue;
	pString:= __NEW(STRING(1), (nLength + 1));
	CONCAT2(pString, pValue, pString, nLength + 1);
ELSE
	// new Length
	nLength:= nLength + nValue;
	// new pointer
	pString:= __NEW(STRING(1), (SIZEOF(STRING(1)) * (nLength + 1)));
	// copy to
	CONCAT2(pOldList, pValue, pString, nLength + 1);
	// delete old
	__DELETE(pOldList);

END_IF
M_Append:= THIS^;
END_METHOD

METHOD PUBLIC M_AppendBOOL  : I_StringBuilder
VAR_INPUT
	Value:			BOOL;
END_VAR
M_Append(BOOL_TO_STRING(Value));
M_AppendBOOL:= THIS^;
END_METHOD

METHOD PUBLIC M_AppendINT : I_StringBuilder
VAR_INPUT
	Value	: LINT;
END_VAR
M_Append(LINT_TO_STRING(Value));
M_AppendINT:= THIS^;
END_METHOD

METHOD PUBLIC M_AppendREAL : I_StringBuilder
VAR_INPUT
	Value:		LREAL;
	Decimals:	SINT;
END_VAR
M_Append(LREAL_TO_FMTSTR(Value, Decimals, TRUE));
M_AppendREAL:= THIS^;
END_METHOD

METHOD PUBLIC M_Contains : BOOL
VAR_INPUT
	Value	: STRING(255);
END_VAR
M_Contains:= M_Find(Value) <> 0;
END_METHOD

METHOD M_Find : UDINT
VAR_INPUT
	Value	: STRING(255);
END_VAR
M_Find:= FIND2(pString, adr(Value));
END_METHOD

METHOD M_Insert : I_StringBuilder
VAR_INPUT
	Position:	UDINT;
	Value:		STRING(255);
END_VAR
VAR
	pValue: 	POINTER TO STRING(1):=ADR(Value);
	nValue:		UDINT:= LEN2(pValue);
	pOldList:	POINTER TO STRING(1):= pString;
END_VAR
IF nLength > Position AND Position <> 0 THEN
	// new Length
	nLength:= nLength + nValue;
	// new pointer
	pString:= __NEW(STRING(1), (SIZEOF(STRING(1)) * (nLength + 1)));
	// insert
	INSERT2(pOldList, pValue, pString, nLength + 1, Position -1);
	// delete old
	__DELETE(pOldList);
END_IF
M_Insert:= THIS^;
END_METHOD

METHOD M_Reset : I_StringBuilder
__DELETE(pString);
nLength:= 0;
M_Reset:= THIS^;
END_METHOD

METHOD M_ToAny : BOOL
VAR_INPUT
	Value:			ANY;
END_VAR
Memset(Value.pValue, 0, DINT_TO_UDINT(Value.diSize));
Memcpy(Value.pValue, pString, nLength + 1);
END_METHOD

METHOD PUBLIC M_ToString : STRING(255)
VAR_INPUT
END_VAR
Memcpy(Adr(M_ToString), pString, nLength + 1);
END_METHOD

PROPERTY PUBLIC P_Length : Udint
GET
P_Length:= nLength;
END_GET
END_PROPERTY

END_FUNCTION_BLOCK

// List/Builder/I_StringBuilder
INTERFACE I_StringBuilder

METHOD M_Append : I_StringBuilder
VAR_INPUT
	Value	: STRING(255);
END_VAR
END_METHOD

METHOD PUBLIC M_AppendBOOL  : I_StringBuilder
VAR_INPUT
	Value:			BOOL;
END_VAR
END_METHOD

METHOD PUBLIC M_AppendINT : I_StringBuilder
VAR_INPUT
	Value	: LINT;
END_VAR
END_METHOD

METHOD PUBLIC M_AppendREAL : I_StringBuilder
VAR_INPUT
	Value:		LREAL;
	Decimals:	SINT;
END_VAR
END_METHOD

METHOD PUBLIC M_Contains : BOOL
VAR_INPUT
	Value	: STRING(255);
END_VAR
END_METHOD

METHOD M_Find : UDINT
VAR_INPUT
	Value	: STRING(255);
END_VAR
END_METHOD

METHOD M_Insert : I_StringBuilder
VAR_INPUT
	Position:	UDINT;
	Value:		STRING(255);
END_VAR
END_METHOD

METHOD M_Reset : I_StringBuilder
END_METHOD

METHOD M_ToAny : BOOL
VAR_INPUT
	Value:			ANY_STRING;
END_VAR
END_METHOD

METHOD PUBLIC M_ToString : String(255)
VAR_INPUT
END_VAR
END_METHOD

PROPERTY PUBLIC P_Length : Udint
GET
END_GET
END_PROPERTY

END_INTERFACE

// Base/F_GetCycleTime
FUNCTION F_GetCycleTime : LREAL
VAR_INPUT
END_VAR
VAR
	fbTask:				GETCURTASKINDEX;
END_VAR

fbTask();
F_GetCycleTime:= UDINT_TO_LREAL(TwinCAT_SystemInfoVarList._TaskInfo[fbTask.index].CycleTime) / 10000000;

END_FUNCTION

// Base/F_GetName
FUNCTION F_GetName : STRING(255)
VAR_INPUT
	InstancePath:		STRING(255);
END_VAR
VAR
    sName:				STRING(255);
    nPosition:			INT;
END_VAR

sName := CONCAT(TwinCAT_SystemInfoVarList._AppInfo.ProjectName, '.');

nPosition := FIND(InstancePath, sName);

IF nPosition > 0 THEN
    F_GetName:= DELETE(InstancePath, nPosition-1 + LEN(sName), 1);
END_IF

nPosition := FIND(F_GetName, sName);

IF nPosition > 0 THEN
    F_GetName:= DELETE(F_GetName, nPosition - 1 + LEN(sName), 1);
END_IF

nPosition:= FIND(STR1 := F_GetName, '.');
F_GetName:= RIGHT(STR := F_GetName, LEN(STR := F_GetName) - nPosition);

END_FUNCTION

// Base/FB_Base
{attribute 'reflection'}
FUNCTION_BLOCK FB_Base IMPLEMENTS I_Base
VAR_INPUT
END_VAR
VAR_OUTPUT
END_VAR
VAR
	{attribute 'instance-path'} 
    {attribute 'noinit'}
    {attribute 'hide'} 
    sInstancePath:		STRING(255);
	eState: 			E_Base;
	eRequest: 			E_Base;
	nState: 			INT;
	{attribute 'hide'} 
	fbGetTime:			NT_GetTime;
	nCycleCount: 		UDINT;
END_VAR

// Prevent double calls
IF nCycleCount <> TwinCAT_SystemInfoVarList._TaskInfo[GETCURTASKINDEXEX()].CycleCount THEN
	nCycleCount:= TwinCAT_SystemInfoVarList._TaskInfo[GETCURTASKINDEXEX()].CycleCount;
	
	fbGetTime();
	
	CASE eState OF
		E_Base.Init:
			IF M_Init() THEN
				eState:= E_Base.Stopped;
				nState:= 0;
			END_IF
			
		E_Base.Stopped:
			IF M_Stopped() THEN
				eState:= E_Base.Starting;
				nState:= 0;
			ELSE
				CASE eRequest OF
					E_Base.Starting, E_Base.Execute:
						eState:= E_Base.Starting;
						nState:= 0;
				END_CASE
			END_IF
			
		E_Base.Starting:
			IF M_Starting() THEN
				eState:= E_Base.Execute;
				nState:= 0;
			END_IF
			
		E_Base.Execute:
			IF M_Execute() THEN
				eState:= E_Base.Stopping;
				nState:= 0;
			ELSE
				CASE eRequest OF
					E_Base.Stopping, E_Base.Stopped:
						eState:= E_Base.Stopping;
						nState:= 0;
				END_CASE
			END_IF
			
		E_Base.Stopping:
			IF M_Stopping() THEN
				eState:= E_Base.Stopped;
				nState:= 0;
			END_IF
	
		E_Base.Aborting:
			IF M_Aborting() THEN
				eState:= E_Base.Aborted;
				nState:= 0;
			END_IF
		
		E_Base.Aborted:
			IF M_Aborted() THEN
				eState:= E_Base.Aborted;
				nState:= 0;
			ELSE
				CASE eRequest OF
					E_Base.Reset:
						eState:= E_Base.Starting;
						nState:= 0;
				END_CASE
			END_IF
			
	END_CASE
	
	eRequest:= eState;
END_IF

METHOD PROTECTED M_Aborted : BOOL
VAR_INPUT
END_VAR
END_METHOD

METHOD PROTECTED M_Aborting : BOOL
VAR_INPUT
END_VAR
END_METHOD

METHOD PROTECTED M_Execute : BOOL
VAR_INPUT
END_VAR
END_METHOD

METHOD PROTECTED M_Init : BOOL
VAR_INPUT
END_VAR
M_Init:= True;
END_METHOD

METHOD M_Request : BOOL
VAR_INPUT
	eState:		E_Base;
END_VAR
eRequest:= eState;
M_Request:= this^.eState = eRequest;
END_METHOD

METHOD PROTECTED M_Starting : BOOL
VAR_INPUT
END_VAR
IF fbGetTime.START THEN
	IF fbGetTime.BUSY THEN
		;
	ELSE
		fbGetTime.START:= FALSE;
		M_Starting:= TRUE;
	END_IF
ELSE
	fbGetTime.START:= TRUE;
END_IF
END_METHOD

METHOD PROTECTED M_Stopped : BOOL
VAR_INPUT
END_VAR
END_METHOD

METHOD PROTECTED M_Stopping : BOOL
VAR_INPUT
END_VAR
M_Stopping:= True;
END_METHOD

PROPERTY PUBLIC P_State : E_Base
GET
P_State:= eState;
END_GET
END_PROPERTY

END_FUNCTION_BLOCK

// Base/I_Base
INTERFACE I_Base EXTENDS I_Object

METHOD M_Request : BOOL
VAR_INPUT
	eState:		E_Base;
END_VAR
END_METHOD

PROPERTY PUBLIC P_State : E_Base
GET
END_GET
END_PROPERTY

END_INTERFACE

// List/Object/I_Object
INTERFACE I_Object EXTENDS __SYSTEM.IQueryInterface

END_INTERFACE

// File/FB_File
{attribute 'no_explicit_call'} 
FUNCTION_BLOCK FB_File
VAR
    fbCreateDir:	FB_CreateDir;
	fbOpen:			FB_FileOpen;
	fbRead:			FB_FileRead;
	fbLoad:			FB_FileLoad;
	fbWrite:		FB_FileWrite;
	fbClose:		FB_FileClose;
	fbDelete:		FB_FileDelete;
END_VAR
VAR_OUTPUT
	eError:			E_AdsError:= E_AdsError.NOERR;
END_VAR

METHOD PUBLIC M_Append : BOOL
VAR_INPUT
	Text:			STRING(255);
END_VAR
fbWrite();
IF fbWrite.bExecute THEN
	IF fbWrite.bError THEN
		eError:= fbWrite.nErrId;
		fbWrite.bExecute:= FALSE;
	ELSIF fbWrite.bBusy THEN
		;
	ELSE
		M_Append:= TRUE;
		fbWrite.bExecute:= FALSE;
	END_IF
ELSE
	fbWrite.bExecute:= TRUE;
	fbWrite.pWriteBuff:= ADR(Text);
	fbWrite.cbWriteLen:= INT_TO_UDINT(Len(Text));
END_IF
END_METHOD

METHOD PUBLIC M_AppendLine : BOOL
VAR_INPUT
	Text:			STRING(255);
END_VAR
Text:= Concat(Text, '$R');
M_AppendLine:= M_Append(Text);
END_METHOD

METHOD PUBLIC M_Close : BOOL
VAR_INPUT
END_VAR
fbClose();
IF fbClose.bExecute THEN
	IF fbClose.hFile = 0 THEN
		fbClose.bExecute:= FALSE;
		M_Close:= TRUE;
	ELSIF fbClose.bError THEN
		fbClose.bExecute:= FALSE;
		eError:= fbClose.nErrId;
	ELSIF fbClose.bBusy THEN
		;
	ELSE
		eError:= E_AdsError.NOERR;	
		fbRead.hFile:= 0;
		fbWrite.hFile:= 0;
		fbClose.hFile:= 0;
		fbClose.bExecute:= FALSE;
		M_Close:= TRUE;
	END_IF
ELSE
	fbClose.bExecute:= TRUE;
END_IF
END_METHOD

METHOD PUBLIC M_Create : BOOL
VAR_INPUT
	PathName:		STRING(255);
END_VAR
VAR
	nTemp: INT;
END_VAR
VAR_INST
	nPosition: INT;
END_VAR
fbCreateDir();
nTemp := FIND(RIGHT(PathName, LEN(PathName) - nPosition), '\');
if nTemp <> 0 then
	IF fbCreateDir.bExecute THEN
		IF NOT fbCreateDir.bBusy THEN
			nPosition := nPosition + nTemp;
			fbCreateDir.bExecute:= FALSE;
		END_IF
	ELSE
		fbCreateDir.bExecute:= TRUE;
		fbCreateDir.ePath:= PATH_GENERIC;
		fbCreateDir.sPathName:= Left(PathName, nPosition + nTemp);
	END_IF
ELSE
	IF M_Open(PathName) THEN
		M_Create:= TRUE;
		nPosition:= 0;
	END_IF
END_IF
END_METHOD

METHOD PUBLIC M_Delete : BOOL
VAR_INPUT
	PathName:		STRING(255);
END_VAR
fbDelete();
IF fbDelete.bExecute THEN
	IF fbDelete.bError THEN
		fbDelete.bExecute:= FALSE;
		M_Delete:= TRUE;
	ELSIF fbDelete.bBusy THEN
		;
	ELSE
		fbDelete.bExecute:= FALSE;
		M_Delete:= TRUE;
	END_IF
ELSE
	fbDelete.bExecute:= TRUE;
	fbDelete.sPathName:= PathName;
	fbDelete.ePath:= E_OpenPath.PATH_GENERIC;
END_IF
END_METHOD

METHOD PUBLIC M_Load : BOOL
VAR_INPUT
	PathName:		STRING(255);
	Value:			ANY;
END_VAR
fbLoad();
IF fbLoad.bExecute THEN
	IF fbLoad.bError THEN
		eError:= fbLoad.nErrId;
		fbLoad.bExecute:= FALSE;
	ELSIF fbLoad.bBusy THEN
		;
	ELSE
		M_Load:= TRUE;
	END_IF
ELSE
	fbLoad.sPathName:= PathName;
	fbLoad.bExecute:= TRUE;
	fbLoad.pReadBuff:= Value.pValue;
	fbLoad.cbReadLen:= DINT_TO_UDINT(Value.diSize);
END_IF
END_METHOD

METHOD PUBLIC M_Open : BOOL
VAR_INPUT
	PathName:		STRING(255);
END_VAR
fbOpen();
IF fbOpen.bExecute THEN
	IF fbOpen.bError THEN
		eError:= fbOpen.nErrId;
		fbOpen.bExecute:= FALSE;
	ELSIF fbOpen.bBusy THEN
		;
	ELSE
		fbRead.hFile:= fbOpen.hFile;
		fbWrite.hFile:= fbOpen.hFile;
		fbClose.hFile:= fbOpen.hFile;
		fbOpen.bExecute:= FALSE;
		M_Open:= TRUE;
	END_IF	
ELSE
	fbOpen.bExecute:= TRUE;
	fbOpen.sPathName:= PathName;
	fbOpen.nMode:= (FOPEN_MODEAPPEND OR FOPEN_MODEPLUS OR FOPEN_MODETEXT);
END_IF
END_METHOD

METHOD PUBLIC M_Read : BOOL
VAR_INPUT
	Value:		ANY;
END_VAR
fbRead();
IF fbRead.bExecute THEN
	IF fbRead.bError THEN
		eError:= fbRead.nErrId;
		fbRead.bExecute:= FALSE;
	ELSIF fbRead.bBusy THEN
		;
	ELSE
		fbRead.bExecute:= FALSE;
		M_Read:= TRUE;
	END_IF
ELSE
	fbRead.bExecute:= TRUE;
	fbRead.pReadBuff:= Value.pValue;
	fbRead.cbReadLen:= DINT_TO_UDINT(Value.diSize);
END_IF
END_METHOD

METHOD PUBLIC M_Write : BOOL
VAR_INPUT
	Value:		ANY;
END_VAR
fbWrite();
IF fbWrite.bExecute THEN
	IF fbWrite.bError THEN
		eError:= fbWrite.nErrId;
		fbWrite.bExecute:= FALSE;
	ELSIF fbWrite.bBusy THEN
		M_Write:= FALSE;
	ELSE
		M_Write:= TRUE;
		fbWrite.bExecute:= FALSE;
	END_IF
ELSE
	fbWrite.bExecute:= TRUE;
	fbRead.pReadBuff:= Value.pValue;
	fbRead.cbReadLen:= DINT_TO_UDINT(Value.diSize);
END_IF
END_METHOD

PROPERTY PUBLIC P_Error : E_AdsError
GET
P_Error:= eError;
END_GET
END_PROPERTY

END_FUNCTION_BLOCK

// File/I_File
INTERFACE I_File

METHOD PUBLIC M_Append : BOOL
VAR_INPUT
	sText:			STRING(255);
END_VAR
END_METHOD

METHOD PUBLIC M_AppendLine : BOOL
VAR_INPUT
	sText:			STRING(255);
END_VAR
END_METHOD

METHOD PUBLIC M_Close : BOOL
VAR_INPUT
END_VAR
END_METHOD

METHOD PUBLIC M_Create : BOOL
VAR_INPUT
	sPathName:		T_MaxString;
END_VAR
END_METHOD

METHOD PUBLIC M_Delete : BOOL
VAR_INPUT
	sPathName:		T_MaxString;
END_VAR
END_METHOD

METHOD PUBLIC M_Load : BOOL
VAR_INPUT
	sPathName:		T_MaxString;
	pData:			PVOID;
	nData:			UDINT;
END_VAR
END_METHOD

METHOD PUBLIC M_Open : BOOL
VAR_INPUT
	sPathName:		T_MaxString;
END_VAR
END_METHOD

METHOD PUBLIC M_Read : BOOL
VAR_INPUT
	Value:		ANY;
END_VAR
END_METHOD

METHOD PUBLIC M_Write : BOOL
VAR_INPUT
	Value:		ANY;
END_VAR
END_METHOD

PROPERTY PUBLIC P_Error : E_AdsError
GET
END_GET
END_PROPERTY

END_INTERFACE

// List/Object/FB_ListObject
{attribute 'no_explicit_call'} 
FUNCTION_BLOCK PUBLIC FB_ListObject IMPLEMENTS I_ListObject
VAR
	pList: 			POINTER TO I_Object;
	nLength:		DINT;
	aList:			POINTER TO POINTER TO ARRAY [0..100] OF I_Object:=ADR(pList);
END_VAR

METHOD FB_exit : BOOL
VAR_INPUT
	bInCopyCode : BOOL; // if TRUE, the exit method is called for exiting an instance that is copied afterwards (online change).
END_VAR
M_Clear();
END_METHOD

METHOD M_Add : BOOL
VAR_INPUT
	Object: 	I_Object;
END_VAR
VAR
	pOldList: 	POINTER TO I_Object;
END_VAR
IF Object <> 0 THEN
	// First Item
	IF pList = 0 THEN
		nLength:= nLength + 1;
		pList:= __NEW(POINTER TO I_Object,DINT_TO_UDINT(nLength));
	ELSE
		// Item already in List
		IF M_Find(Object) = -1 THEN
			// backup 
			pOldList:= pList;
			// new Length
			nLength:= nLength + 1;
			// new pointer
			pList:= __NEW(POINTER TO I_Object,DINT_TO_UDINT(nLength));
			// restore
			Memcpy(pList,pOldList, SIZEOF(POINTER TO I_Object)*DINT_TO_UDINT(nLength -1));
			// delete old
			__DELETE(pOldList);
		ELSE
			M_Add:= FALSE;	
			RETURN;
		END_IF
	END_IF
	IF pList = 0 THEN
		RETURN;
	END_IF
	// add new Object
	pList[nLength-1]:= Object;
	M_Add:= TRUE;
ELSE
	M_Add:= FALSE;	
END_IF
END_METHOD

METHOD M_Clear
IF pList <> 0 THEN
	nLength:= 0;
	__DELETE(pList);
END_IF
END_METHOD

METHOD M_Find : DINT
VAR_INPUT
	Object: 	I_Object;
END_VAR
VAR
	nIndex: 	UINT;
END_VAR
// Object already in List
M_Find := -1;
WHILE nIndex < nLength DO
    IF (pList[nIndex] = Object) THEN
        M_Find := nIndex;
        RETURN;
    END_IF
	nIndex := nIndex + 1;
END_WHILE
END_METHOD

METHOD M_Get : I_Object
VAR_INPUT
	Index: 	DINT;
END_VAR
IF Index <= nLength THEN
	M_Get:= pList[Index];
END_IF
END_METHOD

METHOD M_Index : DINT
VAR_INPUT
	Object: 	I_Object;
END_VAR
VAR
	nIndex: 	DINT;
END_VAR
// Object already in List
M_Index := -1;
WHILE nIndex < nLength DO
    IF (pList[nIndex] = Object) THEN
        M_Index := nIndex;
        RETURN;
    END_IF
	nIndex := nIndex + 1;
END_WHILE
END_METHOD

METHOD M_Remove : BOOL
VAR_INPUT
	Object: 	I_Object;
END_VAR
VAR
	pOldList:			POINTER TO I_Object;
	nPosition: 			DINT;
END_VAR
IF Object <> 0 THEN
	// First Item
	IF nLength >= 0 THEN
		// Item already in List
		nPosition:= M_Find(Object);
		IF nPosition <> -1 THEN
			// backup 
			pOldList:= pList;
			// new Length
			nLength:= nLength -1;
			// new pointer
			pList:= __NEW(POINTER TO I_Object,DINT_TO_UDINT(nLength));
			// restore lower part
			Memcpy(pList,pOldList, SIZEOF(POINTER TO I_Object) * DINT_TO_UDINT(nPosition));
			//pList[nPosition]:= iObject;
			Memcpy(pList + (SIZEOF(POINTER TO I_Object)*nPosition),pOldList + (SIZEOF(POINTER TO I_Object)*(nPosition + 1)), SIZEOF(POINTER TO I_Object) * DINT_TO_UDINT(nLength - nPosition));
			// delete old
			__DELETE(pOldList);
		ELSE
			M_Remove:= FALSE;	
			RETURN;
		END_IF
	ELSE
		M_Remove:= FALSE;	
		RETURN;
	END_IF
	M_Remove:= TRUE;
ELSE
	M_Remove:= FALSE;	
END_IF
END_METHOD

PROPERTY P_Length : DINT
GET
P_Length:= nLength;
END_GET
END_PROPERTY

END_FUNCTION_BLOCK

// List/Object/I_ListObject
INTERFACE I_ListObject

METHOD M_Add : BOOL
VAR_INPUT
	Object: 	I_Object;
END_VAR
END_METHOD

METHOD M_Clear
END_METHOD

METHOD M_Find : DINT
VAR_INPUT
	Object: 	I_Object;
END_VAR
END_METHOD

METHOD M_Get : I_Object
VAR_INPUT
	Index: 	DINT;
END_VAR
END_METHOD

METHOD M_Index : DINT
VAR_INPUT
	Object: 	I_Object;
END_VAR
END_METHOD

METHOD M_Remove : BOOL
VAR_INPUT
	Object: 	I_Object;
END_VAR
END_METHOD

PROPERTY P_Length : DINT
GET
END_GET
END_PROPERTY

END_INTERFACE

// Logger/FB_Logger
{attribute 'no_explicit_call'} 
FUNCTION_BLOCK ABSTRACT FB_Logger IMPLEMENTS I_Logger
VAR_INPUT
END_VAR
VAR_OUTPUT
END_VAR
VAR
	stSettings:		ST_LoggerSettings;
END_VAR

METHOD M_Critical
VAR_INPUT
	Message	: STRING(255);
END_VAR
END_METHOD

METHOD M_Debug
VAR_INPUT
	Message	: STRING(255);
END_VAR
END_METHOD

METHOD M_Error
VAR_INPUT
	Message:		STRING(255);
END_VAR
END_METHOD

METHOD M_Info
VAR_INPUT
	Message	: STRING(255);
END_VAR
END_METHOD

METHOD M_Log
VAR_INPUT
	LogLevel:		E_LogLevel;
	Message:		STRING(255);
END_VAR
END_METHOD

METHOD M_Warning
VAR_INPUT
	Message	: STRING(255);
END_VAR
END_METHOD

{attribute 'suppress_wrn_C0410'}
PROPERTY PUBLIC P_Settings : reference to ST_LoggerSettings
GET
P_Settings ref= stSettings;
END_GET
SET
P_Settings ref= stSettings;
END_SET
END_PROPERTY

END_FUNCTION_BLOCK

// Logger/I_Logger
INTERFACE I_Logger EXTENDS __SYSTEM.IQueryInterface

METHOD M_Critical
VAR_INPUT
	Message:		STRING(255);
END_VAR
END_METHOD

METHOD M_Debug
VAR_INPUT
	Message:		STRING(255);
END_VAR
END_METHOD

METHOD M_Error
VAR_INPUT
	Message:		STRING(255);
END_VAR
END_METHOD

METHOD M_Info
VAR_INPUT
	Message:		STRING(255);
END_VAR
END_METHOD

METHOD M_Log
VAR_INPUT
	LogLevel:		E_LogLevel;
	Message:		STRING(255);
END_VAR
END_METHOD

METHOD M_Warning
VAR_INPUT
	Message:		STRING(255);
END_VAR
END_METHOD

{attribute 'suppress_wrn_C0410'}
PROPERTY PUBLIC P_Settings : reference to ST_LoggerSettings
GET
END_GET
SET
END_SET
END_PROPERTY

END_INTERFACE

// Logger/FB_TcLogger
FUNCTION_BLOCK FB_TcLogger EXTENDS FB_Logger
VAR_INPUT
END_VAR
VAR_OUTPUT
END_VAR
VAR
END_VAR

METHOD M_Critical
VAR_INPUT
	Message:		STRING(255);
END_VAR
M_Log(E_LogLevel.Critical, Message);
END_METHOD

METHOD M_Debug
VAR_INPUT
	Message:		STRING(255);
END_VAR
M_Log(E_LogLevel.Debug, Message);
END_METHOD

METHOD M_Error
VAR_INPUT
	Message:		STRING(255);
END_VAR
M_Log(E_LogLevel.Error, Message);
END_METHOD

METHOD M_Info
VAR_INPUT
	Message:		STRING(255);
END_VAR
M_Log(E_LogLevel.Info, Message);
END_METHOD

METHOD M_Log
VAR_INPUT
	LogLevel:		E_LogLevel;
	Message:		STRING(255);
END_VAR
CASE LogLevel OF
	E_LogLevel.Debug:
		IF LogLevel >= stSettings.eLogLevelMinimum AND LogLevel <= stSettings.eLogLevelMaximum THEN
			ADSLOGSTR(ADSLOG_MSGTYPE_STRING OR ADSLOG_MSGTYPE_LOG,'Debug: %s', Message);
		END_IF
		
	E_LogLevel.Info:
		IF LogLevel >= stSettings.eLogLevelMinimum AND LogLevel <= stSettings.eLogLevelMaximum THEN
			ADSLOGSTR(ADSLOG_MSGTYPE_HINT OR ADSLOG_MSGTYPE_LOG,'Info: %s', Message);
		END_IF
		
	E_LogLevel.Warning:
		IF LogLevel >= stSettings.eLogLevelMinimum AND LogLevel <= stSettings.eLogLevelMaximum THEN
			ADSLOGSTR(ADSLOG_MSGTYPE_WARN OR ADSLOG_MSGTYPE_LOG,'Warning: %s', Message);
		END_IF
		
	E_LogLevel.Error:
		IF LogLevel >= stSettings.eLogLevelMinimum AND LogLevel <= stSettings.eLogLevelMaximum THEN
			ADSLOGSTR(ADSLOG_MSGTYPE_ERROR OR ADSLOG_MSGTYPE_LOG,'Error: %s', Message);
		END_IF
		
	E_LogLevel.Critical:
		IF LogLevel >= stSettings.eLogLevelMinimum AND LogLevel <= stSettings.eLogLevelMaximum THEN
			ADSLOGSTR(ADSLOG_MSGTYPE_ERROR OR ADSLOG_MSGTYPE_LOG,'Critical: %s', Message);
		END_IF
		
END_CASE
END_METHOD

METHOD M_Warning
VAR_INPUT
	Message:		STRING(255);
END_VAR
M_Log(E_LogLevel.Warning, Message);
END_METHOD

{attribute 'suppress_wrn_C0410'}
PROPERTY PUBLIC P_Settings : reference to ST_LoggerSettings
GET
P_Settings ref= stSettings;
END_GET
SET
P_Settings ref= stSettings;
END_SET
END_PROPERTY

END_FUNCTION_BLOCK

// Property/FB_Property
FUNCTION_BLOCK FB_Property IMPLEMENTS I_Property
VAR_INPUT
END_VAR
VAR_OUTPUT
END_VAR
VAR
	fbStringBuilder:	FB_StringBuilder;
	fbList:				FB_ListSTRING;
END_VAR

METHOD PUBLIC M_Add : BOOL
VAR_INPUT
	Name:			STRING(255);
	Value:			STRING(255);
END_VAR
VAR
	nIndex: 		INT;
	sKey:			STRING(255);
END_VAR
fbStringBuilder.M_Reset();
fbStringBuilder.M_Append('<property name="');
fbStringBuilder.M_Append(Name);
sKey:= fbStringBuilder.M_ToString();
fbStringBuilder.M_Append('" value="');
fbStringBuilder.M_Append(Value);
fbStringBuilder.M_Append('" />');

WHILE nIndex < fbList.P_Length DO
	IF FIND(fbList.M_Item(nIndex), sKey) <> 0 THEN
		fbList.M_Set(nIndex, fbStringBuilder.M_ToString());
		RETURN;
	END_IF
	nIndex:= nIndex +1;
END_WHILE
fbList.M_Add(fbStringBuilder.M_ToString());
M_Add:= TRUE;
END_METHOD

METHOD PUBLIC M_Reset
fbStringBuilder.M_Reset();
fbList.M_Clear();
END_METHOD

PROPERTY PUBLIC P_List : I_ListSTRING
GET
P_List:= fbList;
END_GET
END_PROPERTY

END_FUNCTION_BLOCK

// Property/I_Property
INTERFACE I_Property

METHOD PUBLIC M_Add : BOOL
VAR_INPUT
	Name:			STRING(255);
	Value:			STRING(255);
END_VAR
END_METHOD

METHOD PUBLIC M_Reset
END_METHOD

END_INTERFACE

// Testsuite/FB_Testsuite
FUNCTION_BLOCK FB_Testsuite EXTENDS FB_Base IMPLEMENTS I_Testsuite
VAR_INPUT
END_VAR
VAR_OUTPUT
END_VAR
VAR
	stOptions:			ST_TestsuiteOptions;
	stTestsuite:		ST_Testsuite;
	stTestcase:			ST_Testcase;
	nActual:			INT:=  E_Testcase.Init;
	nNext:				INT;
	fCycleTime: 		LREAL;	
	iParent:			I_Testsuites;
	fbTimeout:			TON:= (PT:= T#300S);
	fbRuntime:			TON:= (PT:= T#300S);
	fbBuilder:			FB_StringBuilder;
	fbList:				FB_ListSTRING;
	fbProperty:			FB_Property;
	fbAssert:			FB_Assert;
	iLogger:			I_Logger;
END_VAR

SUPER^();

METHOD PROTECTED M_Execute : BOOL
VAR_INPUT
END_VAR
VAR
	nIndex: DINT:=0;
END_VAR
IF fbTimeout.PT <> T#0S THEN
	fbTimeout(IN:= TRUE);
END_IF
stTestcase.nAssertions:= fbAssert.nAssert;
IF nActual <> nNext THEN
	IF fbAssert.nSkipped <> 0 THEN
			fbBuilder.M_Reset();
			fbBuilder.M_Append('$T$T<testcase name="');
			fbBuilder.M_Append(stTestCase.sName);
			fbBuilder.M_Append('" classname="');
			fbBuilder.M_Append(stTestCase.sClassname);
			fbBuilder.M_Append('" assertions="');
			fbBuilder.M_AppendINT(stTestCase.nAssertions);
			fbBuilder.M_Append('" time="');
			fbBuilder.M_AppendREAL(stTestCase.fTime, 4);
			fbBuilder.M_Append('" file="');
			fbBuilder.M_Append(stTestCase.sFile);
			fbBuilder.M_Append('" line="');
			fbBuilder.M_Append(stTestCase.sLine);
			fbBuilder.M_Append('" >');
			fbList.M_Add(fbBuilder.M_ToString());
			WHILE nIndex < fbAssert.fbList.P_Length DO
				fbList.M_Add(fbAssert.fbList.M_Item(nIndex));
				IF iLogger <> 0 THEN
					iLogger.M_Warning(stTestcase.sName);					
				END_IF
				nIndex:= nIndex + 1;
			END_WHILE
			fbList.M_Add('$T$T</testcase>');
			stTestsuite.nTests:= stTestsuite.nTests + 1;
			stTestsuite.nFailures:= stTestsuite.nFailures + fbAssert.nFailures;
			stTestsuite.nErrors:= stTestsuite.nErrors + fbAssert.nErrors;
			stTestsuite.nSkipped:= stTestsuite.nSkipped + fbAssert.nSkipped;
			stTestsuite.nAssertions:= stTestsuite.nAssertions + fbAssert.nAssert;
			stTestcase.fTime:= 0.0;
			fbTimeout(IN:= FALSE);
			nActual:= nNext;
	ELSIF fbAssert.nPassed = fbAssert.nAssert THEN
		fbBuilder.M_Reset();
		fbBuilder.M_Append('$T$T<testcase name="');
		fbBuilder.M_Append(stTestcase.sName);
		fbBuilder.M_Append('" classname="');
		fbBuilder.M_Append(stTestcase.sClassname);
		fbBuilder.M_Append('" assertions="');
		fbBuilder.M_AppendINT(stTestcase.nAssertions);
		fbBuilder.M_Append('" time="');
		fbBuilder.M_AppendREAL(stTestcase.fTime, 4);
		fbBuilder.M_Append('" file="');
		fbBuilder.M_Append(stTestcase.sFile);
		fbBuilder.M_Append('" line="');
		fbBuilder.M_Append(stTestcase.sLine);
		fbBuilder.M_Append('" />');
		fbList.M_Add(fbBuilder.M_ToString());
	
		stTestsuite.nTests:= stTestsuite.nTests + 1;
		stTestsuite.nFailures:= stTestsuite.nFailures + fbAssert.nFailures;
		stTestsuite.nErrors:= stTestsuite.nErrors + fbAssert.nErrors;
		stTestsuite.nSkipped:= stTestsuite.nSkipped + fbAssert.nSkipped;
		stTestsuite.nAssertions:= stTestsuite.nAssertions + fbAssert.nAssert;
		fbTimeout(IN:= FALSE);
		stTestcase.fTime:= 0.0;
		nActual:= nNext;
	ELSE
		IF fbTimeout.Q THEN
			fbBuilder.M_Reset();
			fbBuilder.M_Append('$T$T<testcase name="');
			fbBuilder.M_Append(stTestCase.sName);
			fbBuilder.M_Append('" classname="');
			fbBuilder.M_Append(stTestCase.sClassname);
			fbBuilder.M_Append('" assertions="');
			fbBuilder.M_AppendINT(stTestCase.nAssertions);
			fbBuilder.M_Append('" time="');
			fbBuilder.M_AppendREAL(stTestCase.fTime, 4);
			fbBuilder.M_Append('" file="');
			fbBuilder.M_Append(stTestCase.sFile);
			fbBuilder.M_Append('" line="');
			fbBuilder.M_Append(stTestCase.sLine);
			fbBuilder.M_Append('" >');
			fbList.M_Add(fbBuilder.M_ToString());
			WHILE nIndex < fbAssert.fbList.P_Length DO
				fbList.M_Add(fbAssert.fbList.M_Item(nIndex));
				IF iLogger <> 0 THEN
					iLogger.M_Error(stTestcase.sName);	
				END_IF
				nIndex:= nIndex + 1;
			END_WHILE
			stTestsuite.nTests:= stTestsuite.nTests + 1;
			stTestsuite.nFailures:= stTestsuite.nFailures + fbAssert.nFailures;
			stTestsuite.nErrors:= stTestsuite.nErrors + fbAssert.nErrors;
			stTestsuite.nSkipped:= stTestsuite.nSkipped + fbAssert.nSkipped;
			stTestsuite.nAssertions:= stTestsuite.nAssertions + fbAssert.nAssert;
			stTestcase.fTime:= 0.0;
			fbTimeout(IN:= FALSE);
			IF stOptions.bAbortOnError THEN
				// Aborted on error in test results
				iLogger.M_Error('Aborted on Error');
				stTestsuite.nFailures:= stTestsuite.nFailures + 1;
				fbList.M_Add('$T$T$T"Aborted on Error"');
				nActual := E_Testcase.Done;
			ELSE
				nActual := nNext;
			END_IF
			fbList.M_Add('$T$T</testcase>');
		END_IF
	END_IF
END_IF
fbRuntime(IN:= TRUE);
stTestsuite.fTime:=  TIME_TO_LREAL(fbRuntime.ET) / 1000.0;
fbAssert.M_Reset();
M_Execute:= nActual = E_Testcase.Done;
END_METHOD

METHOD PROTECTED M_Starting : BOOL
VAR_INPUT
END_VAR

VAR
	nIndex: DINT;
END_VAR
CASE nState OF
	0:
		IF 	SUPER^.M_Starting() THEN
			fbList.M_Clear();
			fbProperty.M_Reset();
			fCycleTime:= F_GetCycleTime();	
			stTestsuite.sName:= F_GetName(sInstancePath);
			stTestsuite.nTests:= 0;
			stTestsuite.nFailures:= 0;		
			stTestsuite.nErrors:= 0;	
			stTestsuite.nSkipped:= 0;		
			stTestsuite.nAssertions:= 0;	
			stTestsuite.fTime:= 0.0;
			stTestsuite.sFile:= '';
			stTestsuite.sTimestamp:= SYSTEMTIME_TO_ISO8601(fbGetTime.TIMESTR, 0, FALSE, 3);
			stTestsuite.sTimestamp:= LEFT(stTestsuite.sTimestamp, LEN(stTestsuite.sTimestamp) - 6);
			nState:= 1;
		END_IF
		
	1:
		nActual:= E_Testcase.Start;
		fbRuntime.IN:= True;
		M_Starting:= TRUE;
	
END_CASE
END_METHOD

METHOD PROTECTED M_Stopping : BOOL
VAR_INPUT
END_VAR
VAR
	sValue: 			STRING(255);
	nIndex: 			DINT:=0;
END_VAR
//    <testsuite name="Tests.Registration" tests="8" failures="1" errors="1" skipped="1" assertions="20" time="16.082687" timestamp="2021-04-02T15:48:23" file="tests/registration.code">
fbBuilder.M_Reset();
fbBuilder.M_Append('$T<testsuite name="');
fbBuilder.M_Append(stTestsuite.sName);
fbBuilder.M_Append('" tests="');
fbBuilder.M_AppendINT(stTestsuite.nTests);
fbBuilder.M_Append('" failures="');
fbBuilder.M_AppendINT(stTestsuite.nFailures);
fbBuilder.M_Append('" errors="');
fbBuilder.M_AppendINT(stTestsuite.nErrors);
fbBuilder.M_Append('" skipped="');
fbBuilder.M_AppendINT(stTestsuite.nSkipped);
fbBuilder.M_Append('" assertions="');
fbBuilder.M_AppendINT(stTestsuite.nAssertions);	
fbBuilder.M_Append('" time="');
fbBuilder.M_AppendREAL(stTestsuite.fTime, 3);
fbBuilder.M_Append('" timestamp="');
fbBuilder.M_Append(stTestsuite.sTimestamp);
fbBuilder.M_Append('" file="');
fbBuilder.M_Append(stTestsuite.sFile);
fbBuilder.M_Append('">');
fbBuilder.M_ToAny(sValue);
fbList.M_Insert(0, sValue);

// add Properties
IF fbProperty.P_List.P_Length > 0 THEN
	fbList.M_Insert(1, '$T$T<properties>');
	nIndex:= 0;
	WHILE nIndex < fbProperty.P_List.P_Length DO
		fbList.M_Insert(2 + nIndex, Concat('$T$T$T', fbProperty.P_List.M_Item(nIndex)));
		nIndex:= nIndex + 1;
	END_WHILE
	fbList.M_Insert(2 + nIndex, '$T$T</properties>');
END_IF

fbList.M_Add('$T</testsuite>');
IF iParent <> 0 THEN
	iParent.P_Data.nTests:= iParent.P_Data.nTests + stTestsuite.nTests;
	iParent.P_Data.nFailures:= iParent.P_Data.nFailures + stTestsuite.nFailures;
	iParent.P_Data.nErrors:= iParent.P_Data.nErrors + stTestsuite.nErrors;
	iParent.P_Data.nSkipped:= iParent.P_Data.nSkipped + stTestsuite.nSkipped;
	iParent.P_Data.nAssertions:= iParent.P_Data.nAssertions + stTestsuite.nAssertions;
	nIndex:= 0;
	WHILE nIndex < fbList.P_Length DO
		iParent.P_List.M_Add(fbList.M_Item(nIndex));
		nIndex:= nIndex + 1;
	END_WHILE
END_IF
fbTimeout(IN:=FALSE);
fbRuntime(IN:=FALSE);
M_Stopping:= TRUE;
END_METHOD

METHOD PUBLIC M_Testcase : BOOL
VAR_INPUT
	Classname:			STRING(255);	// Classname as string
	Timeout:			TIME;			// Timeout as time
	File:				STRING(255);	// File as string
	Line:				STRING(255);	// Line as string
	Next:				INT;			// Next Testcase as int
END_VAR
stTestcase.sName:= CONCAT(CONCAT(CONCAT(stTestsuite.sName,'.'), 'M_Testcase_'), INT_TO_STRING(nActual));
stTestcase.sClassname:= Classname;
stTestcase.nAssertions:= fbAssert.fbList.P_Length;
stTestcase.sFile:= File;
stTestcase.sLine:= Line;
stTestcase.fTime:= stTestcase.fTime + fCycleTime;
fbTimeout.PT:= Timeout;
nNext:= Next;
END_METHOD

PROPERTY PUBLIC P_Assert : I_Assert
GET
P_Assert:= fbAssert;
END_GET
END_PROPERTY

PROPERTY PUBLIC P_File : String(255)
GET
P_File:= stTestsuite.sFile;
END_GET
SET
stTestsuite.sFile:= P_File;
END_SET
END_PROPERTY

PROPERTY PUBLIC P_List : I_ListSTRING
GET
P_List:= fbList;
END_GET
END_PROPERTY

PROPERTY PUBLIC P_Logger : I_Logger
GET
P_Logger:= iLogger;
END_GET
SET
iLogger:= P_Logger;
END_SET
END_PROPERTY

{attribute 'suppress_wrn_C0410'}
PROPERTY PUBLIC P_Options : reference to ST_TestsuiteOptions
GET
P_Options ref= stOptions;
END_GET
SET
P_Options ref= stOptions;
END_SET
END_PROPERTY

PROPERTY PUBLIC P_Parent : I_Testsuites
GET
P_Parent:= iParent;
END_GET
SET
iParent:= P_Parent;
END_SET
END_PROPERTY

PROPERTY PUBLIC P_Property : I_Property
GET
P_Property:= fbProperty;
END_GET
END_PROPERTY

PROPERTY PUBLIC P_Testcase : int
GET
P_Testcase:= nActual;
END_GET
END_PROPERTY

END_FUNCTION_BLOCK

// Testsuite/I_Testsuite
INTERFACE I_Testsuite EXTENDS I_Base

PROPERTY PUBLIC P_File : String(255)
GET
END_GET
SET
END_SET
END_PROPERTY

PROPERTY PUBLIC P_List : I_ListSTRING
GET
END_GET
END_PROPERTY

PROPERTY PUBLIC P_Logger : I_Logger
GET
END_GET
SET
END_SET
END_PROPERTY

{attribute 'suppress_wrn_C0410'}
PROPERTY PUBLIC P_Options : reference to ST_TestsuiteOptions
GET
END_GET
SET
END_SET
END_PROPERTY

PROPERTY PUBLIC P_Parent : I_Testsuites
GET
END_GET
SET
END_SET
END_PROPERTY

PROPERTY PUBLIC P_Testcase : INT
GET
END_GET
END_PROPERTY

END_INTERFACE

// Testsuites/I_Testsuites
INTERFACE I_Testsuites EXTENDS I_Base

{attribute 'suppress_wrn_C0410'}
PROPERTY PUBLIC P_Data : reference to ST_Testsuites
GET
END_GET
SET
END_SET
END_PROPERTY

PROPERTY PUBLIC P_List : I_ListSTRING
GET
END_GET
END_PROPERTY

{attribute 'suppress_wrn_C0410'}
PROPERTY PUBLIC P_Options : REFERENCE TO ST_TestsuitesOptions
GET
END_GET
SET
END_SET
END_PROPERTY

PROPERTY PUBLIC P_Property : I_Property
GET
END_GET
END_PROPERTY

END_INTERFACE

// Testsuites/FB_Testsuites
 FUNCTION_BLOCK PUBLIC FB_Testsuites EXTENDS FB_Base IMPLEMENTS I_Testsuites
VAR_INPUT
END_VAR
VAR_OUTPUT
END_VAR
VAR	
	stOptions:			ST_TestsuitesOptions;
	stTestsuites:    	ST_Testsuites;
	nIndex: 			DINT;
	fbTimeout:			TON:= (PT:= T#300S);
	fbFile:				FB_File;
	fbBuilder:			FB_StringBuilder;
	fbList:				FB_ListSTRING;
	fbListTestsuite:	FB_ListObject;
	fbProperty:			FB_Property;
	fbLogger:			FB_TcLogger;
END_VAR

SUPER^();

METHOD PUBLIC M_Add : BOOL
VAR_INPUT
	Testsuite:		I_Testsuite;
END_VAR
fbListTestsuite.M_Add(Testsuite);
Testsuite.P_Parent:= THIS^;
Testsuite.P_Logger:= fbLogger;
END_METHOD

METHOD PROTECTED M_Execute : BOOL
VAR_INPUT
END_VAR
VAR
	iTestsuite:		I_Testsuite;
	nIndex: 		DINT;
END_VAR
M_Execute:= TRUE;
fbTimeout(IN:= TRUE);
WHILE nIndex < fbListTestsuite.P_Length DO
	IF __QUERYINTERFACE(fbListTestsuite.M_Get(nIndex), iTestsuite) THEN
		M_Execute:= M_Execute AND (iTestsuite.P_State = E_Base.Stopped);
	END_IF
	nIndex:= nIndex + 1;
END_WHILE
IF M_Execute THEN
	stTestsuites.fTime:= TIME_TO_LREAL(fbTimeout.ET) / 1000.0;
	fbTimeout(IN:= FALSE);
END_IF
END_METHOD

METHOD PROTECTED M_Starting : BOOL
VAR_INPUT
END_VAR

VAR
	iTestsuite:		I_Testsuite;
	nIndex: DINT;
END_VAR
CASE nState OF
	0:
		IF 	SUPER^.M_Starting() THEN
			fbList.M_Clear();
			fbProperty.M_Reset();
			stTestsuites.sName:= F_GetName(sInstancePath);
			stTestsuites.nTests:= 0;
			stTestsuites.nFailures:= 0;
			stTestsuites.nErrors:= 0;
			stTestsuites.nSkipped:= 0;
			stTestsuites.nAssertions:= 0;
			stTestsuites.fTime:= 0.0;
			stTestsuites.sTimestamp:= SYSTEMTIME_TO_ISO8601(fbGetTime.TIMESTR, 0, FALSE, 3);
			stTestsuites.sTimestamp:= LEFT(stTestsuites.sTimestamp, LEN(stTestsuites.sTimestamp) - 6);
			nState:= 1;
		END_IF
	
	1:
		WHILE nIndex < fbListTestsuite.P_Length DO
			IF __QUERYINTERFACE(fbListTestsuite.M_Get(nIndex), iTestsuite) THEN
				iTestsuite.M_Request(E_Base.Execute);
			END_IF
			nIndex:= nIndex + 1;
		END_WHILE
		nState:= 2;
		
	2:
		M_Starting:= TRUE;
		
END_CASE
END_METHOD

METHOD PROTECTED M_Stopping : BOOL
VAR_INPUT
END_VAR
VAR
	sValue: STRING(255);
END_VAR
CASE nState OF
	0:
		//<testsuites name="Test run" tests="8" failures="1" errors="1" skipped="1"  assertions="20" time="16.082687" timestamp="2021-04-02T15:48:23">
		fbList.M_Insert(0, '<?xml version="1.0" encoding="UTF-8"?>');
		fbBuilder.M_Reset();
		fbBuilder.M_Append('<testsuites name="');	
		fbBuilder.M_Append(stTestsuites.sName);		
		fbBuilder.M_Append('" tests="');	
		fbBuilder.M_AppendINT(stTestsuites.nTests);
		fbBuilder.M_Append('" failures="');	
		fbBuilder.M_AppendINT(stTestsuites.nFailures);
		fbBuilder.M_Append('" errors="');	
		fbBuilder.M_AppendINT(stTestsuites.nErrors);
		fbBuilder.M_Append('" skipped="');	
		fbBuilder.M_AppendINT(stTestsuites.nSkipped);
		fbBuilder.M_Append('" assertions="');	
		fbBuilder.M_AppendINT(stTestsuites.nAssertions);
		fbBuilder.M_Append('" time="');	
		fbBuilder.M_AppendREAL(stTestsuites.fTime, 3);
		fbBuilder.M_Append('" timestamp="');
		fbBuilder.M_Append(stTestsuites.sTimestamp);
		fbBuilder.M_Append('">');
		fbBuilder.M_ToAny(sValue);
		fbList.M_Insert(1, sValue);
		fbList.M_Add('</testsuites>');
		nState:= 1;
	1:	
		// add Properties
		IF fbProperty.P_List.P_Length > 0 THEN
			fbList.M_Insert(2, '$T<properties>');
			nIndex:= 0;
			WHILE nIndex < fbProperty.P_List.P_Length DO
				fbList.M_Insert(3 + nIndex, Concat('$T$T', fbProperty.P_List.M_Item(nIndex)));
				nIndex:= nIndex + 1;
			END_WHILE
			fbList.M_Insert(3 + nIndex, '$T</properties>');
		END_IF
		nState:= 2;
		
	2:
		fbBuilder.M_Reset();
		fbBuilder.M_Append(stTestsuites.sName);		
		fbBuilder.M_Append(': tests= ');
		fbBuilder.M_AppendINT(stTestsuites.nTests);
		fbBuilder.M_Append(' failures= ');	
		fbBuilder.M_AppendINT(stTestsuites.nFailures);
		fbBuilder.M_Append(' errors= ');	
		fbBuilder.M_AppendINT(stTestsuites.nErrors);
		fbBuilder.M_Append(' skipped= ');	
		fbBuilder.M_AppendINT(stTestsuites.nSkipped);
		fbBuilder.M_Append(' assertions= ');
		fbBuilder.M_AppendINT(stTestsuites.nAssertions);
		fbBuilder.M_ToAny(sValue);
		IF stTestsuites.nFailures <> 0 OR_ELSE stTestsuites.nErrors <> 0 THEN
			fbLogger.M_Error(sValue);
		ELSIF stTestsuites.nSkipped <> 0 THEN
			fbLogger.M_Warning(sValue);
		ELSE
			fbLogger.M_Info(sValue);
		END_IF
		nState:= 3;
			
	3:
		IF fbFile.M_Delete(stOptions.sFilePathName) THEN
			nState:= 4;
		END_IF	
	
	4:
		IF fbFile.M_Create(stOptions.sFilePathName) THEN
			nState:= 5;
			nIndex:= 0;
		END_IF
	
	5:
			IF fbFile.M_AppendLine(fbList.M_Item(nIndex)) THEN
				IF nIndex > fbList.P_Length THEN
					nState:= 6;
				END_IF
				nIndex:= nIndex +1;
			END_IF	
	6:
		M_Stopping:= fbFile.M_Close();	
		
END_CASE
END_METHOD

{attribute 'suppress_wrn_C0410'}
PROPERTY PUBLIC P_Data : reference to ST_Testsuites
GET
P_Data ref= stTestsuites;
END_GET
SET
P_Data ref= stTestsuites;
END_SET
END_PROPERTY

PROPERTY PUBLIC P_List : I_ListSTRING
GET
P_List:= fbList;
END_GET
END_PROPERTY

{attribute 'suppress_wrn_C0410'}
PROPERTY PUBLIC P_Options : REFERENCE TO ST_TestsuitesOptions
GET
P_Options ref= stOptions;
END_GET
SET
P_Options ref= stOptions;
END_SET
END_PROPERTY

PROPERTY PUBLIC P_Property : I_Property
GET
P_Property:= fbProperty;
END_GET
END_PROPERTY

END_FUNCTION_BLOCK
